LIN {X 0,Y 624.93,Z 1040.405,A -85,B 0,C 180,E1 29774.882,E2 29774.882} C_VEL
LIN {X 0,Y 625.518,Z 1029.116,A -85,B 0,C 180,E1 29772.895,E2 29772.895} C_VEL
LIN {X 0,Y 626.333,Z 1016.12,A -85,B 0,C 180,E1 29770.897,E2 29770.897} C_VEL
LIN {X 0,Y 627.354,Z 1001.616,A -85,B 0,C 180,E1 29768.985,E2 29768.985} C_VEL
LIN {X 0,Y 628.562,Z 986,A -85,B 0,C 180,E1 29767.161,E2 29767.161} C_VEL
LIN {X 0,Y 629.943,Z 968.823,A -85,B 0,C 180,E1 29765.426,E2 29765.426} C_VEL
LIN {X 0,Y 631.502,Z 950.498,A -85,B 0,C 180,E1 29763.784,E2 29763.784} C_VEL
LIN {X 0,Y 633.079,Z 931.694,A -85,B 0,C 180,E1 29762.332,E2 29762.332} C_VEL
LIN {X 0,Y 634.609,Z 913.191,A -85,B 0,C 180,E1 29761.072,E2 29761.072} C_VEL
LIN {X 0,Y 636.354,Z 890.919,A -85,B 0,C 180,E1 29759.762,E2 29759.762} C_VEL
LIN {X 0,Y 637.792,Z 871.802,A -85,B 0,C 180,E1 29758.793,E2 29758.793} C_VEL
LIN {X 0,Y 639.438,Z 848.234,A -85,B 0,C 180,E1 29757.776,E2 29757.776} C_VEL
LIN {X 0,Y 640.692,Z 827.149,A -85,B 0,C 180,E1 29757.025,E2 29757.025} C_VEL
LIN {X 0,Y 641.942,Z 803.825,A -85,B 0,C 180,E1 29756.343,E2 29756.343} C_VEL
LIN {X 0,Y 642.944,Z 779.718,A -85,B 0,C 180,E1 29755.822,E2 29755.822} C_VEL
LIN {X 0,Y 643.646,Z 755.972,A -85,B 0,C 180,E1 29755.448,E2 29755.448} C_VEL
LIN {X 0,Y 647.272,Z 508.069,A -85,B 0,C 180,E1 29752.341,E2 29752.341} C_VEL
LIN {X 0,Y 648.694,Z 406.811,A -85,B 0,C 180,E1 29751.044,E2 29751.044} C_VEL
LIN {X 0,Y 643.579,Z 386.076,A -85,B 0,C 180,E1 29750.391,E2 29750.391} C_VEL
LIN {X 0,Y 636.999,Z 374.634,A -85,B 0,C 180,E1 29749.718,E2 29749.718} C_VEL
LIN {X 0,Y 630.181,Z 356.926,A -85,B 0,C 180,E1 29747.68,E2 29747.68} C_VEL
LIN {X 0,Y 625.657,Z 345.944,A -85,B 0,C 180,E1 29746.338,E2 29746.338} C_VEL
LIN {X 0,Y 624.887,Z 343.395,A -85,B 0,C 180,E1 29746.017,E2 29746.017} C_VEL
LIN {X 0,Y 624.953,Z 343.388,A -85,B 0,C 180,E1 29742.967,E2 29742.967} C_VEL
LIN {X 0,Y 624.886,Z 343.382,A -85,B 0,C 180,E1 29739.963,E2 29739.963} C_VEL
LIN {X 0,Y 624.956,Z 343.376,A -85,B 0,C 180,E1 29736.983,E2 29736.983} C_VEL
LIN {X 0,Y 624.887,Z 343.383,A -85,B 0,C 180,E1 29733.948,E2 29733.948} C_VEL
LIN {X 0,Y 624.955,Z 343.374,A -85,B 0,C 180,E1 29730.903,E2 29730.903} C_VEL
LIN {X 0,Y 624.889,Z 343.378,A -85,B 0,C 180,E1 29727.855,E2 29727.855} C_VEL
LIN {X 0,Y 624.956,Z 343.385,A -85,B 0,C 180,E1 29724.783,E2 29724.783} C_VEL
LIN {X 0,Y 624.887,Z 343.388,A -85,B 0,C 180,E1 29721.791,E2 29721.791} C_VEL
LIN {X 0,Y 624.939,Z 343.372,A -85,B 0,C 180,E1 29718.856,E2 29718.856} C_VEL
LIN {X 0,Y 624.891,Z 343.384,A -85,B 0,C 180,E1 29715.784,E2 29715.784} C_VEL
LIN {X 0,Y 624.92,Z 343.379,A -85,B 0,C 180,E1 29712.944,E2 29712.944} C_VEL
LIN {X 0,Y 624.894,Z 343.373,A -85,B 0,C 180,E1 29709.765,E2 29709.765} C_VEL
LIN {X 0,Y 624.915,Z 343.385,A -85,B 0,C 180,E1 29706.892,E2 29706.892} C_VEL
LIN {X 0,Y 624.896,Z 343.383,A -85,B 0,C 180,E1 29703.67,E2 29703.67} C_VEL
LIN {X 0,Y 624.912,Z 343.384,A -85,B 0,C 180,E1 29700.825,E2 29700.825} C_VEL
LIN {X 0,Y 624.9,Z 343.389,A -85,B 0,C 180,E1 29697.616,E2 29697.616} C_VEL
LIN {X 0,Y 624.907,Z 343.379,A -85,B 0,C 180,E1 29694.767,E2 29694.767} C_VEL
LIN {X 0,Y 624.903,Z 343.389,A -85,B 0,C 180,E1 29691.535,E2 29691.535} C_VEL
LIN {X 0,Y 624.908,Z 343.369,A -85,B 0,C 180,E1 29688.65,E2 29688.65} C_VEL
LIN {X 0,Y 624.904,Z 343.384,A -85,B 0,C 180,E1 29685.451,E2 29685.451} C_VEL
LIN {X 0,Y 624.907,Z 343.38,A -85,B 0,C 180,E1 29682.59,E2 29682.59} C_VEL
LIN {X 0,Y 624.906,Z 343.375,A -85,B 0,C 180,E1 29679.389,E2 29679.389} C_VEL
LIN {X 0,Y 624.899,Z 343.386,A -85,B 0,C 180,E1 29676.62,E2 29676.62} C_VEL
LIN {X 0,Y 624.918,Z 343.387,A -85,B 0,C 180,E1 29673.384,E2 29673.384} C_VEL
LIN {X 0,Y 624.895,Z 343.374,A -85,B 0,C 180,E1 29670.578,E2 29670.578} C_VEL
LIN {X 0,Y 624.941,Z 343.379,A -85,B 0,C 180,E1 29667.478,E2 29667.478} C_VEL
LIN {X 0,Y 624.896,Z 343.387,A -85,B 0,C 180,E1 29664.491,E2 29664.491} C_VEL
LIN {X 0,Y 624.937,Z 343.387,A -85,B 0,C 180,E1 29661.333,E2 29661.333} C_VEL
LIN {X 0,Y 624.896,Z 343.391,A -85,B 0,C 180,E1 29658.391,E2 29658.391} C_VEL
LIN {X 0,Y 624.934,Z 343.351,A -85,B 0,C 180,E1 29655.251,E2 29655.251} C_VEL
LIN {X 0,Y 624.894,Z 343.384,A -85,B 0,C 180,E1 29652.333,E2 29652.333} C_VEL
LIN {X 0,Y 624.953,Z 343.473,A -85,B 0,C 180,E1 29649.73,E2 29649.73} C_VEL
LIN {X 0,Y 626.203,Z 346.794,A -85,B 0,C 180,E1 29649.306,E2 29649.306} C_VEL
LIN {X 0,Y 627.768,Z 350.392,A -85,B 0,C 180,E1 29648.961,E2 29648.961} C_VEL
LIN {X 0,Y 629.852,Z 356.916,A -85,B 0,C 180,E1 29648.631,E2 29648.631} C_VEL
LIN {X 0,Y 633.845,Z 372.513,A -85,B 0,C 180,E1 29648.1,E2 29648.1} C_VEL
LIN {X 0,Y 635.947,Z 377.186,A -85,B 0,C 180,E1 29647.875,E2 29647.875} C_VEL
LIN {X 0,Y 642.615,Z 388.681,A -85,B 0,C 180,E1 29647.223,E2 29647.223} C_VEL
LIN {X 0,Y 638.708,Z 628.744,A -85,B 0,C 180,E1 29644.159,E2 29644.159} C_VEL
LIN {X 0,Y 636.879,Z 738.868,A -85,B 0,C 180,E1 29642.751,E2 29642.751} C_VEL
LIN {X 0,Y 635.934,Z 764.323,A -85,B 0,C 180,E1 29642.266,E2 29642.266} C_VEL
LIN {X 0,Y 634.929,Z 784.357,A -85,B 0,C 180,E1 29641.755,E2 29641.755} C_VEL
LIN {X 0,Y 633.679,Z 806.259,A -85,B 0,C 180,E1 29641.063,E2 29641.063} C_VEL
LIN {X 0,Y 631.998,Z 829.361,A -85,B 0,C 180,E1 29640.154,E2 29640.154} C_VEL
LIN {X 0,Y 630.445,Z 849.976,A -85,B 0,C 180,E1 29639.189,E2 29639.189} C_VEL
LIN {X 0,Y 628.6,Z 871.75,A -85,B 0,C 180,E1 29637.985,E2 29637.985} C_VEL
LIN {X 0,Y 626.972,Z 889.893,A -85,B 0,C 180,E1 29636.829,E2 29636.829} C_VEL
LIN {X 0,Y 625.011,Z 910.955,A -85,B 0,C 180,E1 29635.287,E2 29635.287} C_VEL
LIN {X 0,Y 623.503,Z 927.172,A -85,B 0,C 180,E1 29633.923,E2 29633.923} C_VEL
LIN {X 0,Y 621.814,Z 945.972,A -85,B 0,C 180,E1 29632.146,E2 29632.146} C_VEL
LIN {X 0,Y 620.415,Z 962.253,A -85,B 0,C 180,E1 29630.372,E2 29630.372} C_VEL
LIN {X 0,Y 619.163,Z 977.823,A -85,B 0,C 180,E1 29628.453,E2 29628.453} C_VEL
LIN {X 0,Y 618.189,Z 991.221,A -85,B 0,C 180,E1 29626.539,E2 29626.539} C_VEL
LIN {X 0,Y 617.383,Z 1004.094,A -85,B 0,C 180,E1 29624.443,E2 29624.443} C_VEL
LIN {X 0,Y 616.791,Z 1014.91,A -85,B 0,C 180,E1 29622.356,E2 29622.356} C_VEL
LIN {X 0,Y 616.386,Z 1024.556,A -85,B 0,C 180,E1 29620.184,E2 29620.184} C_VEL
LIN {X 0,Y 616.118,Z 1032.294,A -85,B 0,C 180,E1 29618.023,E2 29618.023} C_VEL
LIN {X 0,Y 616.001,Z 1038.045,A -85,B 0,C 180,E1 29616.056,E2 29616.056} C_VEL
LIN {X 0,Y 615.93,Z 1043.189,A -85,B 0,C 180,E1 29613.723,E2 29613.723} C_VEL
LIN {X 0,Y 615.915,Z 1046.127,A -85,B 0,C 180,E1 29611.768,E2 29611.768} C_VEL
LIN {X 0,Y 615.9,Z 1048.037,A -85,B 0,C 180,E1 29609.628,E2 29609.628} C_VEL
LIN {X 0,Y 615.894,Z 1048.372,A -85,B 0,C 180,E1 29607.395,E2 29607.395} C_VEL
LIN {X 0,Y 615.9,Z 1047.414,A -85,B 0,C 180,E1 29605.423,E2 29605.423} C_VEL
LIN {X 0,Y 615.92,Z 1044.749,A -85,B 0,C 180,E1 29603.1,E2 29603.1} C_VEL
LIN {X 0,Y 615.961,Z 1040.849,A -85,B 0,C 180,E1 29601.035,E2 29601.035} C_VEL
LIN {X 0,Y 616.051,Z 1035.367,A -85,B 0,C 180,E1 29598.864,E2 29598.864} C_VEL
LIN {X 0,Y 616.246,Z 1028.13,A -85,B 0,C 180,E1 29596.679,E2 29596.679} C_VEL
LIN {X 0,Y 616.539,Z 1020.478,A -85,B 0,C 180,E1 29594.768,E2 29594.768} C_VEL
LIN {X 0,Y 617.068,Z 1009.43,A -85,B 0,C 180,E1 29592.459,E2 29592.459} C_VEL
LIN {X 0,Y 617.72,Z 998.488,A -85,B 0,C 180,E1 29590.522,E2 29590.522} C_VEL
LIN {X 0,Y 618.662,Z 984.485,A -85,B 0,C 180,E1 29588.377,E2 29588.377} C_VEL
LIN {X 0,Y 619.676,Z 971.194,A -85,B 0,C 180,E1 29586.613,E2 29586.613} C_VEL
LIN {X 0,Y 621.016,Z 955.276,A -85,B 0,C 180,E1 29584.743,E2 29584.743} C_VEL
LIN {X 0,Y 622.444,Z 938.805,A -85,B 0,C 180,E1 29583.063,E2 29583.063} C_VEL
LIN {X 0,Y 624.226,Z 919.692,A -85,B 0,C 180,E1 29581.332,E2 29581.332} C_VEL
LIN {X 0,Y 625.918,Z 901.36,A -85,B 0,C 180,E1 29579.894,E2 29579.894} C_VEL
LIN {X 0,Y 627.697,Z 882.047,A -85,B 0,C 180,E1 29578.554,E2 29578.554} C_VEL
LIN {X 0,Y 629.506,Z 861.113,A -85,B 0,C 180,E1 29577.313,E2 29577.313} C_VEL
LIN {X 0,Y 631.175,Z 840.831,A -85,B 0,C 180,E1 29576.273,E2 29576.273} C_VEL
LIN {X 0,Y 632.919,Z 817.134,A -85,B 0,C 180,E1 29575.256,E2 29575.256} C_VEL
LIN {X 0,Y 634.242,Z 796.202,A -85,B 0,C 180,E1 29574.511,E2 29574.511} C_VEL
LIN {X 0,Y 635.639,Z 770.4,A -85,B 0,C 180,E1 29573.785,E2 29573.785} C_VEL
LIN {X 0,Y 636.544,Z 749.103,A -85,B 0,C 180,E1 29573.334,E2 29573.334} C_VEL
LIN {X 0,Y 637.275,Z 721.539,A -85,B 0,C 180,E1 29572.919,E2 29572.919} C_VEL
LIN {X 0,Y 641.355,Z 468.268,A -85,B 0,C 180,E1 29569.706,E2 29569.706} C_VEL
LIN {X 0,Y 642.577,Z 388.154,A -85,B 0,C 180,E1 29568.66,E2 29568.66} C_VEL
LIN {X 0,Y 628.337,Z 364.446,A -85,B 0,C 180,E1 29567.206,E2 29567.206} C_VEL
LIN {X 0,Y 619.079,Z 350.106,A -85,B 0,C 180,E1 29566.217,E2 29566.217} C_VEL
LIN {X 0,Y 616.951,Z 344.375,A -85,B 0,C 180,E1 29565.432,E2 29565.432} C_VEL
LIN {X 0,Y 617.017,Z 344.368,A -85,B 0,C 180,E1 29562.357,E2 29562.357} C_VEL
LIN {X 0,Y 616.95,Z 344.369,A -85,B 0,C 180,E1 29559.323,E2 29559.323} C_VEL
LIN {X 0,Y 617.011,Z 344.339,A -85,B 0,C 180,E1 29556.264,E2 29556.264} C_VEL
LIN {X 0,Y 616.951,Z 344.377,A -85,B 0,C 180,E1 29553.216,E2 29553.216} C_VEL
LIN {X 0,Y 617.02,Z 344.373,A -85,B 0,C 180,E1 29550.077,E2 29550.077} C_VEL
LIN {X 0,Y 616.953,Z 344.377,A -85,B 0,C 180,E1 29547.092,E2 29547.092} C_VEL
LIN {X 0,Y 617.012,Z 344.374,A -85,B 0,C 180,E1 29543.938,E2 29543.938} C_VEL
LIN {X 0,Y 616.95,Z 344.37,A -85,B 0,C 180,E1 29540.988,E2 29540.988} C_VEL
LIN {X 0,Y 617.016,Z 344.363,A -85,B 0,C 180,E1 29537.933,E2 29537.933} C_VEL
LIN {X 0,Y 616.95,Z 344.375,A -85,B 0,C 180,E1 29534.933,E2 29534.933} C_VEL
LIN {X 0,Y 617.015,Z 344.374,A -85,B 0,C 180,E1 29531.877,E2 29531.877} C_VEL
LIN {X 0,Y 616.949,Z 344.372,A -85,B 0,C 180,E1 29528.857,E2 29528.857} C_VEL
LIN {X 0,Y 617.016,Z 344.362,A -85,B 0,C 180,E1 29525.86,E2 29525.86} C_VEL
LIN {X 0,Y 616.948,Z 344.376,A -85,B 0,C 180,E1 29522.787,E2 29522.787} C_VEL
LIN {X 0,Y 617.023,Z 344.375,A -85,B 0,C 180,E1 29519.721,E2 29519.721} C_VEL
LIN {X 0,Y 616.947,Z 344.366,A -85,B 0,C 180,E1 29516.655,E2 29516.655} C_VEL
LIN {X 0,Y 617.018,Z 344.361,A -85,B 0,C 180,E1 29513.58,E2 29513.58} C_VEL
LIN {X 0,Y 616.949,Z 344.376,A -85,B 0,C 180,E1 29510.579,E2 29510.579} C_VEL
LIN {X 0,Y 617.014,Z 344.368,A -85,B 0,C 180,E1 29507.553,E2 29507.553} C_VEL
LIN {X 0,Y 616.947,Z 344.364,A -85,B 0,C 180,E1 29504.489,E2 29504.489} C_VEL
LIN {X 0,Y 617.015,Z 344.364,A -85,B 0,C 180,E1 29501.443,E2 29501.443} C_VEL
LIN {X 0,Y 616.948,Z 344.376,A -85,B 0,C 180,E1 29498.414,E2 29498.414} C_VEL
LIN {X 0,Y 617.003,Z 344.37,A -85,B 0,C 180,E1 29495.489,E2 29495.489} C_VEL
LIN {X 0,Y 616.951,Z 344.371,A -85,B 0,C 180,E1 29492.385,E2 29492.385} C_VEL
LIN {X 0,Y 616.989,Z 344.378,A -85,B 0,C 180,E1 29489.519,E2 29489.519} C_VEL
LIN {X 0,Y 616.953,Z 344.378,A -85,B 0,C 180,E1 29486.339,E2 29486.339} C_VEL
LIN {X 0,Y 616.991,Z 344.377,A -85,B 0,C 180,E1 29483.389,E2 29483.389} C_VEL
LIN {X 0,Y 616.956,Z 344.379,A -85,B 0,C 180,E1 29480.316,E2 29480.316} C_VEL
LIN {X 0,Y 616.969,Z 344.367,A -85,B 0,C 180,E1 29477.483,E2 29477.483} C_VEL
LIN {X 0,Y 617.023,Z 344.531,A -85,B 0,C 180,E1 29474.692,E2 29474.692} C_VEL
LIN {X 0,Y 625.556,Z 365.763,A -85,B 0,C 180,E1 29471.99,E2 29471.99} C_VEL
LIN {X 0,Y 629.163,Z 375.222,A -85,B 0,C 180,E1 29470.899,E2 29470.899} C_VEL
LIN {X 0,Y 638.485,Z 391.346,A -85,B 0,C 180,E1 29469.935,E2 29469.935} C_VEL
LIN {X 0,Y 642.629,Z 410.143,A -85,B 0,C 180,E1 29469.355,E2 29469.355} C_VEL
LIN {X 0,Y 638.25,Z 677.094,A -85,B 0,C 180,E1 29465.951,E2 29465.951} C_VEL
LIN {X 0,Y 636.738,Z 767.252,A -85,B 0,C 180,E1 29464.797,E2 29464.797} C_VEL
LIN {X 0,Y 635.766,Z 792.504,A -85,B 0,C 180,E1 29464.317,E2 29464.317} C_VEL
LIN {X 0,Y 634.738,Z 812.614,A -85,B 0,C 180,E1 29463.808,E2 29463.808} C_VEL
LIN {X 0,Y 633.457,Z 835.069,A -85,B 0,C 180,E1 29463.103,E2 29463.103} C_VEL
LIN {X 0,Y 631.844,Z 857.447,A -85,B 0,C 180,E1 29462.229,E2 29462.229} C_VEL
LIN {X 0,Y 630.335,Z 877.622,A -85,B 0,C 180,E1 29461.299,E2 29461.299} C_VEL
LIN {X 0,Y 628.484,Z 900.405,A -85,B 0,C 180,E1 29460.062,E2 29460.062} C_VEL
LIN {X 0,Y 626.885,Z 918.89,A -85,B 0,C 180,E1 29458.9,E2 29458.9} C_VEL
LIN {X 0,Y 625.021,Z 939.869,A -85,B 0,C 180,E1 29457.392,E2 29457.392} C_VEL
LIN {X 0,Y 623.487,Z 957.138,A -85,B 0,C 180,E1 29455.964,E2 29455.964} C_VEL
LIN {X 0,Y 621.967,Z 974.396,A -85,B 0,C 180,E1 29454.353,E2 29454.353} C_VEL
LIN {X 0,Y 620.503,Z 991.086,A -85,B 0,C 180,E1 29452.552,E2 29452.552} C_VEL
LIN {X 0,Y 619.292,Z 1006.237,A -85,B 0,C 180,E1 29450.707,E2 29450.707} C_VEL
LIN {X 0,Y 618.235,Z 1020.607,A -85,B 0,C 180,E1 29448.677,E2 29448.677} C_VEL
LIN {X 0,Y 617.432,Z 1033.123,A -85,B 0,C 180,E1 29446.657,E2 29446.657} C_VEL
LIN {X 0,Y 616.82,Z 1044.181,A -85,B 0,C 180,E1 29444.552,E2 29444.552} C_VEL
LIN {X 0,Y 616.445,Z 1052.774,A -85,B 0,C 180,E1 29442.649,E2 29442.649} C_VEL
LIN {X 0,Y 616.144,Z 1061.604,A -85,B 0,C 180,E1 29440.283,E2 29440.283} C_VEL
LIN {X 0,Y 616.019,Z 1067.49,A -85,B 0,C 180,E1 29438.306,E2 29438.306} C_VEL
LIN {X 0,Y 615.943,Z 1072.696,A -85,B 0,C 180,E1 29436.057,E2 29436.057} C_VEL
LIN {X 0,Y 615.908,Z 1076.01,A -85,B 0,C 180,E1 29433.91,E2 29433.91} C_VEL
LIN {X 0,Y 615.905,Z 1077.836,A -85,B 0,C 180,E1 29431.954,E2 29431.954} C_VEL
LIN {X 0,Y 615.895,Z 1078.417,A -85,B 0,C 180,E1 29429.628,E2 29429.628} C_VEL
LIN {X 0,Y 615.909,Z 1077.495,A -85,B 0,C 180,E1 29427.581,E2 29427.581} C_VEL
LIN {X 0,Y 615.921,Z 1075.085,A -85,B 0,C 180,E1 29425.344,E2 29425.344} C_VEL
LIN {X 0,Y 615.947,Z 1071.102,A -85,B 0,C 180,E1 29423.194,E2 29423.194} C_VEL
LIN {X 0,Y 616.023,Z 1066.219,A -85,B 0,C 180,E1 29421.224,E2 29421.224} C_VEL
LIN {X 0,Y 616.234,Z 1058.661,A -85,B 0,C 180,E1 29418.867,E2 29418.867} C_VEL
LIN {X 0,Y 616.531,Z 1050.749,A -85,B 0,C 180,E1 29416.876,E2 29416.876} C_VEL
LIN {X 0,Y 617.024,Z 1040.404,A -85,B 0,C 180,E1 29414.684,E2 29414.684} C_VEL
LIN {X 0,Y 617.67,Z 1029.115,A -85,B 0,C 180,E1 29412.671,E2 29412.671} C_VEL
LIN {X 0,Y 618.548,Z 1016.119,A -85,B 0,C 180,E1 29410.647,E2 29410.647} C_VEL
LIN {X 0,Y 619.65,Z 1001.614,A -85,B 0,C 180,E1 29408.711,E2 29408.711} C_VEL
LIN {X 0,Y 620.977,Z 985.782,A -85,B 0,C 180,E1 29406.842,E2 29406.842} C_VEL
LIN {X 0,Y 622.442,Z 968.822,A -85,B 0,C 180,E1 29405.11,E2 29405.11} C_VEL
LIN {X 0,Y 623.88,Z 952.658,A -85,B 0,C 180,E1 29403.644,E2 29403.644} C_VEL
LIN {X 0,Y 625.655,Z 932.82,A -85,B 0,C 180,E1 29402.079,E2 29402.079} C_VEL
LIN {X 0,Y 627.208,Z 915.193,A -85,B 0,C 180,E1 29400.855,E2 29400.855} C_VEL
LIN {X 0,Y 629.064,Z 893.416,A -85,B 0,C 180,E1 29399.533,E2 29399.533} C_VEL
LIN {X 0,Y 630.661,Z 873.465,A -85,B 0,C 180,E1 29398.499,E2 29398.499} C_VEL
LIN {X 0,Y 632.318,Z 851.795,A -85,B 0,C 180,E1 29397.53,E2 29397.53} C_VEL
LIN {X 0,Y 633.817,Z 828.417,A -85,B 0,C 180,E1 29396.675,E2 29396.675} C_VEL
LIN {X 0,Y 635.037,Z 807.046,A -85,B 0,C 180,E1 29396.035,E2 29396.035} C_VEL
LIN {X 0,Y 636.223,Z 781.484,A -85,B 0,C 180,E1 29395.452,E2 29395.452} C_VEL
LIN {X 0,Y 636.947,Z 759.346,A -85,B 0,C 180,E1 29395.09,E2 29395.09} C_VEL
LIN {X 0,Y 640.743,Z 518.127,A -85,B 0,C 180,E1 29392.034,E2 29392.034} C_VEL
LIN {X 0,Y 642.4,Z 408.639,A -85,B 0,C 180,E1 29390.624,E2 29390.624} C_VEL
LIN {X 0,Y 637.907,Z 390.365,A -85,B 0,C 180,E1 29390.04,E2 29390.04} C_VEL
LIN {X 0,Y 628.778,Z 374.728,A -85,B 0,C 180,E1 29389.126,E2 29389.126} C_VEL
LIN {X 0,Y 620.891,Z 354.378,A -85,B 0,C 180,E1 29386.711,E2 29386.711} C_VEL
LIN {X 0,Y 616.988,Z 344.415,A -85,B 0,C 180,E1 29385.47,E2 29385.47} C_VEL
LIN {X 0,Y 616.953,Z 344.382,A -85,B 0,C 180,E1 29382.267,E2 29382.267} C_VEL
LIN {X 0,Y 616.974,Z 344.369,A -85,B 0,C 180,E1 29379.442,E2 29379.442} C_VEL
LIN {X 0,Y 616.959,Z 344.381,A -85,B 0,C 180,E1 29376.267,E2 29376.267} C_VEL
LIN {X 0,Y 616.967,Z 344.37,A -85,B 0,C 180,E1 29373.422,E2 29373.422} C_VEL
LIN {X 0,Y 616.959,Z 344.375,A -85,B 0,C 180,E1 29370.16,E2 29370.16} C_VEL
LIN {X 0,Y 616.964,Z 344.364,A -85,B 0,C 180,E1 29367.362,E2 29367.362} C_VEL
LIN {X 0,Y 616.962,Z 344.366,A -85,B 0,C 180,E1 29364.105,E2 29364.105} C_VEL
LIN {X 0,Y 616.964,Z 344.374,A -85,B 0,C 180,E1 29361.27,E2 29361.27} C_VEL
LIN {X 0,Y 616.961,Z 344.376,A -85,B 0,C 180,E1 29357.949,E2 29357.949} C_VEL
LIN {X 0,Y 616.976,Z 344.369,A -85,B 0,C 180,E1 29355.029,E2 29355.029} C_VEL
LIN {X 0,Y 616.957,Z 344.377,A -85,B 0,C 180,E1 29351.783,E2 29351.783} C_VEL
LIN {X 0,Y 616.981,Z 344.358,A -85,B 0,C 180,E1 29348.856,E2 29348.856} C_VEL
LIN {X 0,Y 616.956,Z 344.369,A -85,B 0,C 180,E1 29345.674,E2 29345.674} C_VEL
LIN {X 0,Y 616.99,Z 344.368,A -85,B 0,C 180,E1 29342.694,E2 29342.694} C_VEL
LIN {X 0,Y 616.953,Z 344.359,A -85,B 0,C 180,E1 29339.525,E2 29339.525} C_VEL
LIN {X 0,Y 616.993,Z 344.373,A -85,B 0,C 180,E1 29336.562,E2 29336.562} C_VEL
LIN {X 0,Y 616.952,Z 344.369,A -85,B 0,C 180,E1 29333.392,E2 29333.392} C_VEL
LIN {X 0,Y 616.992,Z 344.373,A -85,B 0,C 180,E1 29330.485,E2 29330.485} C_VEL
LIN {X 0,Y 616.956,Z 344.377,A -85,B 0,C 180,E1 29327.33,E2 29327.33} C_VEL
LIN {X 0,Y 616.979,Z 344.368,A -85,B 0,C 180,E1 29324.49,E2 29324.49} C_VEL
LIN {X 0,Y 616.961,Z 344.377,A -85,B 0,C 180,E1 29321.283,E2 29321.283} C_VEL
LIN {X 0,Y 616.977,Z 344.362,A -85,B 0,C 180,E1 29318.415,E2 29318.415} C_VEL
LIN {X 0,Y 616.959,Z 344.363,A -85,B 0,C 180,E1 29315.173,E2 29315.173} C_VEL
LIN {X 0,Y 616.987,Z 344.374,A -85,B 0,C 180,E1 29312.233,E2 29312.233} C_VEL
LIN {X 0,Y 616.961,Z 344.379,A -85,B 0,C 180,E1 29309.086,E2 29309.086} C_VEL
LIN {X 0,Y 616.988,Z 344.363,A -85,B 0,C 180,E1 29306.118,E2 29306.118} C_VEL
LIN {X 0,Y 616.958,Z 344.372,A -85,B 0,C 180,E1 29302.922,E2 29302.922} C_VEL
LIN {X 0,Y 616.984,Z 344.368,A -85,B 0,C 180,E1 29300.045,E2 29300.045} C_VEL
LIN {X 0,Y 616.958,Z 344.354,A -85,B 0,C 180,E1 29296.828,E2 29296.828} C_VEL
LIN {X 0,Y 617.003,Z 344.371,A -85,B 0,C 180,E1 29293.787,E2 29293.787} C_VEL
LIN {X 0,Y 616.958,Z 344.381,A -85,B 0,C 180,E1 29290.656,E2 29290.656} C_VEL
LIN {X 0,Y 616.962,Z 344.424,A -85,B 0,C 180,E1 29290.312,E2 29290.312} C_VEL
LIN {X 0,Y 619.286,Z 350.473,A -85,B 0,C 180,E1 29289.559,E2 29289.559} C_VEL
LIN {X 0,Y 635.41,Z 376.25,A -85,B 0,C 180,E1 29287.929,E2 29287.929} C_VEL
LIN {X 0,Y 635.947,Z 377.186,A -85,B 0,C 180,E1 29287.875,E2 29287.875} C_VEL
LIN {X 0,Y 637.696,Z 381.876,A -85,B 0,C 180,E1 29287.678,E2 29287.678} C_VEL
LIN {X 0,Y 638.342,Z 388.319,A -85,B 0,C 180,E1 29287.539,E2 29287.539} C_VEL
LIN {X 0,Y 637.479,Z 398.608,A -85,B 0,C 180,E1 29287.456,E2 29287.456} C_VEL
LIN {X 0,Y 636.01,Z 411.557,A -85,B 0,C 180,E1 29287.379,E2 29287.379} C_VEL
LIN {X 0,Y 635.973,Z 412.733,A -85,B 0,C 180,E1 29287.365,E2 29287.365} C_VEL
LIN {X 0,Y 631.746,Z 660.219,A -85,B 0,C 180,E1 29284.189,E2 29284.189} C_VEL
LIN {X 0,Y 630.304,Z 739.834,A -85,B 0,C 180,E1 29283.154,E2 29283.154} C_VEL
LIN {X 0,Y 629.304,Z 764.933,A -85,B 0,C 180,E1 29282.668,E2 29282.668} C_VEL
LIN {X 0,Y 628.251,Z 784.817,A -85,B 0,C 180,E1 29282.156,E2 29282.156} C_VEL
LIN {X 0,Y 626.858,Z 807.75,A -85,B 0,C 180,E1 29281.419,E2 29281.419} C_VEL
LIN {X 0,Y 625.122,Z 830.21,A -85,B 0,C 180,E1 29280.52,E2 29280.52} C_VEL
LIN {X 0,Y 623.405,Z 851.74,A -85,B 0,C 180,E1 29279.499,E2 29279.499} C_VEL
LIN {X 0,Y 621.518,Z 872.423,A -85,B 0,C 180,E1 29278.333,E2 29278.333} C_VEL
LIN {X 0,Y 619.797,Z 890.524,A -85,B 0,C 180,E1 29277.165,E2 29277.165} C_VEL
LIN {X 0,Y 617.646,Z 912.113,A -85,B 0,C 180,E1 29275.558,E2 29275.558} C_VEL
LIN {X 0,Y 616.012,Z 928.638,A -85,B 0,C 180,E1 29274.144,E2 29274.144} C_VEL
LIN {X 0,Y 614.23,Z 946.758,A -85,B 0,C 180,E1 29272.386,E2 29272.386} C_VEL
LIN {X 0,Y 612.691,Z 963.333,A -85,B 0,C 180,E1 29270.541,E2 29270.541} C_VEL
LIN {X 0,Y 611.24,Z 980.108,A -85,B 0,C 180,E1 29268.404,E2 29268.404} C_VEL
LIN {X 0,Y 610.279,Z 992.662,A -85,B 0,C 180,E1 29266.564,E2 29266.564} C_VEL
LIN {X 0,Y 609.399,Z 1005.783,A -85,B 0,C 180,E1 29264.345,E2 29264.345} C_VEL
LIN {X 0,Y 608.841,Z 1015.497,A -85,B 0,C 180,E1 29262.424,E2 29262.424} C_VEL
LIN {X 0,Y 608.41,Z 1025.019,A -85,B 0,C 180,E1 29260.224,E2 29260.224} C_VEL
LIN {X 0,Y 608.139,Z 1032.381,A -85,B 0,C 180,E1 29258.129,E2 29258.129} C_VEL
LIN {X 0,Y 608.012,Z 1038.118,A -85,B 0,C 180,E1 29256.136,E2 29256.136} C_VEL
LIN {X 0,Y 607.934,Z 1043.234,A -85,B 0,C 180,E1 29253.772,E2 29253.772} C_VEL
LIN {X 0,Y 607.916,Z 1046.159,A -85,B 0,C 180,E1 29251.791,E2 29251.791} C_VEL
LIN {X 0,Y 607.901,Z 1048.057,A -85,B 0,C 180,E1 29249.623,E2 29249.623} C_VEL
LIN {X 0,Y 607.894,Z 1048.365,A -85,B 0,C 180,E1 29247.36,E2 29247.36} C_VEL
LIN {X 0,Y 607.899,Z 1047.404,A -85,B 0,C 180,E1 29245.377,E2 29245.377} C_VEL
LIN {X 0,Y 607.921,Z 1044.704,A -85,B 0,C 180,E1 29243.009,E2 29243.009} C_VEL
LIN {X 0,Y 607.97,Z 1040.79,A -85,B 0,C 180,E1 29240.916,E2 29240.916} C_VEL
LIN {X 0,Y 608.075,Z 1035.293,A -85,B 0,C 180,E1 29238.716,E2 29238.716} C_VEL
LIN {X 0,Y 608.286,Z 1028.026,A -85,B 0,C 180,E1 29236.502,E2 29236.502} C_VEL
LIN {X 0,Y 608.599,Z 1020.359,A -85,B 0,C 180,E1 29234.564,E2 29234.564} C_VEL
LIN {X 0,Y 609.176,Z 1009.276,A -85,B 0,C 180,E1 29232.224,E2 29232.224} C_VEL
LIN {X 0,Y 609.848,Z 998.896,A -85,B 0,C 180,E1 29230.36,E2 29230.36} C_VEL
LIN {X 0,Y 610.811,Z 985.692,A -85,B 0,C 180,E1 29228.287,E2 29228.287} C_VEL
LIN {X 0,Y 611.938,Z 971.742,A -85,B 0,C 180,E1 29226.402,E2 29226.402} C_VEL
LIN {X 0,Y 613.377,Z 955.934,A -85,B 0,C 180,E1 29224.51,E2 29224.51} C_VEL
LIN {X 0,Y 615.013,Z 938.663,A -85,B 0,C 180,E1 29222.711,E2 29222.711} C_VEL
LIN {X 0,Y 616.794,Z 921.137,A -85,B 0,C 180,E1 29221.093,E2 29221.093} C_VEL
LIN {X 0,Y 618.683,Z 901.859,A -85,B 0,C 180,E1 29219.558,E2 29219.558} C_VEL
LIN {X 0,Y 620.572,Z 882.575,A -85,B 0,C 180,E1 29218.205,E2 29218.205} C_VEL
LIN {X 0,Y 622.515,Z 861.552,A -85,B 0,C 180,E1 29216.945,E2 29216.945} C_VEL
LIN {X 0,Y 624.171,Z 842.465,A -85,B 0,C 180,E1 29215.952,E2 29215.952} C_VEL
LIN {X 0,Y 626.019,Z 819.2,A -85,B 0,C 180,E1 29214.928,E2 29214.928} C_VEL
LIN {X 0,Y 627.409,Z 798.552,A -85,B 0,C 180,E1 29214.177,E2 29214.177} C_VEL
LIN {X 0,Y 628.81,Z 774.942,A -85,B 0,C 180,E1 29213.476,E2 29213.476} C_VEL
LIN {X 0,Y 629.874,Z 751.394,A -85,B 0,C 180,E1 29212.958,E2 29212.958} C_VEL
LIN {X 0,Y 630.648,Z 727.106,A -85,B 0,C 180,E1 29212.57,E2 29212.57} C_VEL
LIN {X 0,Y 635.022,Z 474.062,A -85,B 0,C 180,E1 29209.328,E2 29209.328} C_VEL
LIN {X 0,Y 636.398,Z 391.316,A -85,B 0,C 180,E1 29208.238,E2 29208.238} C_VEL
LIN {X 0,Y 623.168,Z 369.368,A -85,B 0,C 180,E1 29206.858,E2 29206.858} C_VEL
LIN {X 0,Y 612.17,Z 352.556,A -85,B 0,C 180,E1 29205.66,E2 29205.66} C_VEL
LIN {X 0,Y 610.765,Z 350.187,A -85,B 0,C 180,E1 29205.477,E2 29205.477} C_VEL
LIN {X 0,Y 609.052,Z 345.365,A -85,B 0,C 180,E1 29204.803,E2 29204.803} C_VEL
LIN {X 0,Y 609.018,Z 345.347,A -85,B 0,C 180,E1 29201.667,E2 29201.667} C_VEL
LIN {X 0,Y 609.049,Z 345.361,A -85,B 0,C 180,E1 29198.719,E2 29198.719} C_VEL
LIN {X 0,Y 609.014,Z 345.33,A -85,B 0,C 180,E1 29195.535,E2 29195.535} C_VEL
LIN {X 0,Y 609.056,Z 345.365,A -85,B 0,C 180,E1 29192.58,E2 29192.58} C_VEL
LIN {X 0,Y 609.018,Z 345.364,A -85,B 0,C 180,E1 29189.4,E2 29189.4} C_VEL
LIN {X 0,Y 609.062,Z 345.365,A -85,B 0,C 180,E1 29186.417,E2 29186.417} C_VEL
LIN {X 0,Y 609.017,Z 345.365,A -85,B 0,C 180,E1 29183.308,E2 29183.308} C_VEL
LIN {X 0,Y 609.054,Z 345.361,A -85,B 0,C 180,E1 29180.368,E2 29180.368} C_VEL
LIN {X 0,Y 609.013,Z 345.36,A -85,B 0,C 180,E1 29177.149,E2 29177.149} C_VEL
LIN {X 0,Y 609.066,Z 345.353,A -85,B 0,C 180,E1 29174.159,E2 29174.159} C_VEL
LIN {X 0,Y 609.015,Z 345.363,A -85,B 0,C 180,E1 29171.075,E2 29171.075} C_VEL
LIN {X 0,Y 609.069,Z 345.365,A -85,B 0,C 180,E1 29168.021,E2 29168.021} C_VEL
LIN {X 0,Y 609.01,Z 345.359,A -85,B 0,C 180,E1 29164.898,E2 29164.898} C_VEL
LIN {X 0,Y 609.068,Z 345.352,A -85,B 0,C 180,E1 29161.882,E2 29161.882} C_VEL
LIN {X 0,Y 609.012,Z 345.365,A -85,B 0,C 180,E1 29158.777,E2 29158.777} C_VEL
LIN {X 0,Y 609.075,Z 345.361,A -85,B 0,C 180,E1 29155.669,E2 29155.669} C_VEL
LIN {X 0,Y 609.008,Z 345.352,A -85,B 0,C 180,E1 29152.598,E2 29152.598} C_VEL
LIN {X 0,Y 609.075,Z 345.351,A -85,B 0,C 180,E1 29149.53,E2 29149.53} C_VEL
LIN {X 0,Y 609.01,Z 345.366,A -85,B 0,C 180,E1 29146.421,E2 29146.421} C_VEL
LIN {X 0,Y 609.077,Z 345.357,A -85,B 0,C 180,E1 29143.402,E2 29143.402} C_VEL
LIN {X 0,Y 609.007,Z 345.352,A -85,B 0,C 180,E1 29140.331,E2 29140.331} C_VEL
LIN {X 0,Y 609.082,Z 345.35,A -85,B 0,C 180,E1 29137.307,E2 29137.307} C_VEL
LIN {X 0,Y 609.01,Z 345.366,A -85,B 0,C 180,E1 29134.209,E2 29134.209} C_VEL
LIN {X 0,Y 609.077,Z 345.361,A -85,B 0,C 180,E1 29131.045,E2 29131.045} C_VEL
LIN {X 0,Y 609.009,Z 345.367,A -85,B 0,C 180,E1 29128.084,E2 29128.084} C_VEL
LIN {X 0,Y 609.076,Z 345.363,A -85,B 0,C 180,E1 29125.003,E2 29125.003} C_VEL
LIN {X 0,Y 609.008,Z 345.366,A -85,B 0,C 180,E1 29121.998,E2 29121.998} C_VEL
LIN {X 0,Y 609.08,Z 345.362,A -85,B 0,C 180,E1 29118.896,E2 29118.896} C_VEL
LIN {X 0,Y 609.011,Z 345.369,A -85,B 0,C 180,E1 29115.847,E2 29115.847} C_VEL
LIN {X 0,Y 609.071,Z 345.565,A -85,B 0,C 180,E1 29115.328,E2 29115.328} C_VEL
LIN {X 0,Y 617.648,Z 366.692,A -85,B 0,C 180,E1 29112.558,E2 29112.558} C_VEL
LIN {X 0,Y 620.898,Z 374.872,A -85,B 0,C 180,E1 29111.58,E2 29111.58} C_VEL
LIN {X 0,Y 632.845,Z 395.363,A -85,B 0,C 180,E1 29110.311,E2 29110.311} C_VEL
LIN {X 0,Y 636.439,Z 411.894,A -85,B 0,C 180,E1 29109.793,E2 29109.793} C_VEL
LIN {X 0,Y 631.746,Z 678.208,A -85,B 0,C 180,E1 29106.362,E2 29106.362} C_VEL
LIN {X 0,Y 630.151,Z 767.053,A -85,B 0,C 180,E1 29105.214,E2 29105.214} C_VEL
LIN {X 0,Y 629.116,Z 792.394,A -85,B 0,C 180,E1 29104.729,E2 29104.729} C_VEL
LIN {X 0,Y 628.015,Z 812.716,A -85,B 0,C 180,E1 29104.21,E2 29104.21} C_VEL
LIN {X 0,Y 626.572,Z 836.174,A -85,B 0,C 180,E1 29103.46,E2 29103.46} C_VEL
LIN {X 0,Y 624.875,Z 858.359,A -85,B 0,C 180,E1 29102.578,E2 29102.578} C_VEL
LIN {X 0,Y 623.131,Z 880.429,A -85,B 0,C 180,E1 29101.541,E2 29101.541} C_VEL
LIN {X 0,Y 621.251,Z 901.593,A -85,B 0,C 180,E1 29100.356,E2 29100.356} C_VEL
LIN {X 0,Y 619.546,Z 920.145,A -85,B 0,C 180,E1 29099.17,E2 29099.17} C_VEL
LIN {X 0,Y 617.49,Z 941.596,A -85,B 0,C 180,E1 29097.588,E2 29097.588} C_VEL
LIN {X 0,Y 615.939,Z 958.032,A -85,B 0,C 180,E1 29096.203,E2 29096.203} C_VEL
LIN {X 0,Y 614.202,Z 976.677,A -85,B 0,C 180,E1 29094.425,E2 29094.425} C_VEL
LIN {X 0,Y 612.845,Z 991.46,A -85,B 0,C 180,E1 29092.804,E2 29092.804} C_VEL
LIN {X 0,Y 611.522,Z 1006.997,A -85,B 0,C 180,E1 29090.882,E2 29090.882} C_VEL
LIN {X 0,Y 610.387,Z 1021.24,A -85,B 0,C 180,E1 29088.827,E2 29088.827} C_VEL
LIN {X 0,Y 609.532,Z 1033.689,A -85,B 0,C 180,E1 29086.781,E2 29086.781} C_VEL
LIN {X 0,Y 608.878,Z 1044.639,A -85,B 0,C 180,E1 29084.649,E2 29084.649} C_VEL
LIN {X 0,Y 608.463,Z 1053.583,A -85,B 0,C 180,E1 29082.624,E2 29082.624} C_VEL
LIN {X 0,Y 608.158,Z 1061.907,A -85,B 0,C 180,E1 29080.324,E2 29080.324} C_VEL
LIN {X 0,Y 608.023,Z 1067.491,A -85,B 0,C 180,E1 29078.416,E2 29078.416} C_VEL
LIN {X 0,Y 607.945,Z 1072.696,A -85,B 0,C 180,E1 29076.137,E2 29076.137} C_VEL
LIN {X 0,Y 607.909,Z 1076.009,A -85,B 0,C 180,E1 29073.961,E2 29073.961} C_VEL
LIN {X 0,Y 607.906,Z 1077.836,A -85,B 0,C 180,E1 29071.979,E2 29071.979} C_VEL
LIN {X 0,Y 607.895,Z 1078.417,A -85,B 0,C 180,E1 29069.623,E2 29069.623} C_VEL
LIN {X 0,Y 607.908,Z 1077.495,A -85,B 0,C 180,E1 29067.549,E2 29067.549} C_VEL
LIN {X 0,Y 607.923,Z 1075.085,A -85,B 0,C 180,E1 29065.283,E2 29065.283} C_VEL
LIN {X 0,Y 607.957,Z 1071.102,A -85,B 0,C 180,E1 29063.104,E2 29063.104} C_VEL
LIN {X 0,Y 608.035,Z 1066.219,A -85,B 0,C 180,E1 29061.108,E2 29061.108} C_VEL
LIN {X 0,Y 608.266,Z 1058.66,A -85,B 0,C 180,E1 29058.719,E2 29058.719} C_VEL
LIN {X 0,Y 608.588,Z 1050.748,A -85,B 0,C 180,E1 29056.702,E2 29056.702} C_VEL
LIN {X 0,Y 609.123,Z 1040.402,A -85,B 0,C 180,E1 29054.48,E2 29054.48} C_VEL
LIN {X 0,Y 609.827,Z 1029.113,A -85,B 0,C 180,E1 29052.441,E2 29052.441} C_VEL
LIN {X 0,Y 610.779,Z 1016.117,A -85,B 0,C 180,E1 29050.391,E2 29050.391} C_VEL
LIN {X 0,Y 611.957,Z 1001.612,A -85,B 0,C 180,E1 29048.43,E2 29048.43} C_VEL
LIN {X 0,Y 613.372,Z 985.999,A -85,B 0,C 180,E1 29046.562,E2 29046.562} C_VEL
LIN {X 0,Y 614.907,Z 968.972,A -85,B 0,C 180,E1 29044.813,E2 29044.813} C_VEL
LIN {X 0,Y 616.661,Z 950.759,A -85,B 0,C 180,E1 29043.155,E2 29043.155} C_VEL
LIN {X 0,Y 618.487,Z 931.255,A -85,B 0,C 180,E1 29041.621,E2 29041.621} C_VEL
LIN {X 0,Y 620.297,Z 912.013,A -85,B 0,C 180,E1 29040.286,E2 29040.286} C_VEL
LIN {X 0,Y 622.247,Z 890.482,A -85,B 0,C 180,E1 29039.002,E2 29039.002} C_VEL
LIN {X 0,Y 623.869,Z 871.366,A -85,B 0,C 180,E1 29038.015,E2 29038.015} C_VEL
LIN {X 0,Y 625.724,Z 847.82,A -85,B 0,C 180,E1 29036.982,E2 29036.982} C_VEL
LIN {X 0,Y 627.182,Z 825.971,A -85,B 0,C 180,E1 29036.193,E2 29036.193} C_VEL
LIN {X 0,Y 628.648,Z 801.827,A -85,B 0,C 180,E1 29035.49,E2 29035.49} C_VEL
LIN {X 0,Y 629.71,Z 779.15,A -85,B 0,C 180,E1 29034.997,E2 29034.997} C_VEL
LIN {X 0,Y 630.482,Z 755.478,A -85,B 0,C 180,E1 29034.619,E2 29034.619} C_VEL
LIN {X 0,Y 634.576,Z 507.829,A -85,B 0,C 180,E1 29031.462,E2 29031.462} C_VEL
LIN {X 0,Y 636.13,Z 410.472,A -85,B 0,C 180,E1 29030.196,E2 29030.196} C_VEL
LIN {X 0,Y 632.258,Z 394.616,A -85,B 0,C 180,E1 29029.682,E2 29029.682} C_VEL
LIN {X 0,Y 620.448,Z 374.384,A -85,B 0,C 180,E1 29028.467,E2 29028.467} C_VEL
LIN {X 0,Y 612.728,Z 354.981,A -85,B 0,C 180,E1 29026.089,E2 29026.089} C_VEL
LIN {X 0,Y 609.065,Z 345.367,A -85,B 0,C 180,E1 29024.867,E2 29024.867} C_VEL
LIN {X 0,Y 609.009,Z 345.37,A -85,B 0,C 180,E1 29021.93,E2 29021.93} C_VEL
LIN {X 0,Y 609.077,Z 345.362,A -85,B 0,C 180,E1 29018.837,E2 29018.837} C_VEL
LIN {X 0,Y 609.012,Z 345.368,A -85,B 0,C 180,E1 29015.767,E2 29015.767} C_VEL
LIN {X 0,Y 609.057,Z 345.366,A -85,B 0,C 180,E1 29012.58,E2 29012.58} C_VEL
LIN {X 0,Y 609.014,Z 345.363,A -85,B 0,C 180,E1 29009.616,E2 29009.616} C_VEL
LIN {X 0,Y 609.062,Z 345.353,A -85,B 0,C 180,E1 29006.522,E2 29006.522} C_VEL
LIN {X 0,Y 609.009,Z 345.353,A -85,B 0,C 180,E1 29003.616,E2 29003.616} C_VEL
LIN {X 0,Y 609.076,Z 345.362,A -85,B 0,C 180,E1 29000.568,E2 29000.568} C_VEL
LIN {X 0,Y 609.011,Z 345.364,A -85,B 0,C 180,E1 28997.485,E2 28997.485} C_VEL
LIN {X 0,Y 609.07,Z 345.348,A -85,B 0,C 180,E1 28994.353,E2 28994.353} C_VEL
LIN {X 0,Y 609.012,Z 345.364,A -85,B 0,C 180,E1 28991.363,E2 28991.363} C_VEL
LIN {X 0,Y 609.064,Z 345.355,A -85,B 0,C 180,E1 28988.211,E2 28988.211} C_VEL
LIN {X 0,Y 609.012,Z 345.356,A -85,B 0,C 180,E1 28985.275,E2 28985.275} C_VEL
LIN {X 0,Y 609.069,Z 345.364,A -85,B 0,C 180,E1 28982.164,E2 28982.164} C_VEL
LIN {X 0,Y 609.011,Z 345.346,A -85,B 0,C 180,E1 28979.153,E2 28979.153} C_VEL
LIN {X 0,Y 609.068,Z 345.363,A -85,B 0,C 180,E1 28976.046,E2 28976.046} C_VEL
LIN {X 0,Y 609.014,Z 345.357,A -85,B 0,C 180,E1 28973.022,E2 28973.022} C_VEL
LIN {X 0,Y 609.06,Z 345.352,A -85,B 0,C 180,E1 28969.883,E2 28969.883} C_VEL
LIN {X 0,Y 609.016,Z 345.364,A -85,B 0,C 180,E1 28966.905,E2 28966.905} C_VEL
LIN {X 0,Y 609.062,Z 345.349,A -85,B 0,C 180,E1 28963.794,E2 28963.794} C_VEL
LIN {X 0,Y 609.017,Z 345.363,A -85,B 0,C 180,E1 28960.83,E2 28960.83} C_VEL
LIN {X 0,Y 609.072,Z 345.357,A -85,B 0,C 180,E1 28957.714,E2 28957.714} C_VEL
LIN {X 0,Y 609.013,Z 345.35,A -85,B 0,C 180,E1 28954.731,E2 28954.731} C_VEL
LIN {X 0,Y 609.064,Z 345.357,A -85,B 0,C 180,E1 28951.57,E2 28951.57} C_VEL
LIN {X 0,Y 609.017,Z 345.366,A -85,B 0,C 180,E1 28948.621,E2 28948.621} C_VEL
LIN {X 0,Y 609.065,Z 345.36,A -85,B 0,C 180,E1 28945.5,E2 28945.5} C_VEL
LIN {X 0,Y 609.018,Z 345.364,A -85,B 0,C 180,E1 28942.466,E2 28942.466} C_VEL
LIN {X 0,Y 609.061,Z 345.36,A -85,B 0,C 180,E1 28939.326,E2 28939.326} C_VEL
LIN {X 0,Y 609.015,Z 345.332,A -85,B 0,C 180,E1 28936.389,E2 28936.389} C_VEL
LIN {X 0,Y 609.059,Z 345.368,A -85,B 0,C 180,E1 28933.203,E2 28933.203} C_VEL
LIN {X 0,Y 609.062,Z 345.576,A -85,B 0,C 180,E1 28930.887,E2 28930.887} C_VEL
LIN {X 0,Y 611.013,Z 350.763,A -85,B 0,C 180,E1 28930.235,E2 28930.235} C_VEL
LIN {X 0,Y 626.828,Z 375.591,A -85,B 0,C 180,E1 28928.59,E2 28928.59} C_VEL
LIN {X 0,Y 636.341,Z 391.797,A -85,B 0,C 180,E1 28927.637,E2 28927.637} C_VEL
LIN {X 0,Y 635.973,Z 412.733,A -85,B 0,C 180,E1 28927.365,E2 28927.365} C_VEL
LIN {X 0,Y 635.047,Z 420.433,A -85,B 0,C 180,E1 28927.323,E2 28927.323} C_VEL
LIN {X 0,Y 629.815,Z 441.007,A -85,B 0,C 180,E1 28927.413,E2 28927.413} C_VEL
LIN {X 0,Y 629.133,Z 447.61,A -85,B 0,C 180,E1 28927.368,E2 28927.368} C_VEL
LIN {X 0,Y 624.619,Z 699.187,A -85,B 0,C 180,E1 28924.124,E2 28924.124} C_VEL
LIN {X 0,Y 623.697,Z 743.497,A -85,B 0,C 180,E1 28923.524,E2 28923.524} C_VEL
LIN {X 0,Y 622.627,Z 767.01,A -85,B 0,C 180,E1 28923.044,E2 28923.044} C_VEL
LIN {X 0,Y 621.497,Z 787.189,A -85,B 0,C 180,E1 28922.51,E2 28922.51} C_VEL
LIN {X 0,Y 619.803,Z 812.008,A -85,B 0,C 180,E1 28921.676,E2 28921.676} C_VEL
LIN {X 0,Y 618.178,Z 832.167,A -85,B 0,C 180,E1 28920.847,E2 28920.847} C_VEL
LIN {X 0,Y 616.198,Z 855.203,A -85,B 0,C 180,E1 28919.718,E2 28919.718} C_VEL
LIN {X 0,Y 614.304,Z 874.686,A -85,B 0,C 180,E1 28918.59,E2 28918.59} C_VEL
LIN {X 0,Y 612.292,Z 894.753,A -85,B 0,C 180,E1 28917.262,E2 28917.262} C_VEL
LIN {X 0,Y 610.169,Z 914.461,A -85,B 0,C 180,E1 28915.738,E2 28915.738} C_VEL
LIN {X 0,Y 608.261,Z 932.973,A -85,B 0,C 180,E1 28914.11,E2 28914.11} C_VEL
LIN {X 0,Y 606.372,Z 950.537,A -85,B 0,C 180,E1 28912.32,E2 28912.32} C_VEL
LIN {X 0,Y 604.843,Z 966.182,A -85,B 0,C 180,E1 28910.516,E2 28910.516} C_VEL
LIN {X 0,Y 603.374,Z 981.698,A -85,B 0,C 180,E1 28908.452,E2 28908.452} C_VEL
LIN {X 0,Y 602.275,Z 995.359,A -85,B 0,C 180,E1 28906.393,E2 28906.393} C_VEL
LIN {X 0,Y 601.407,Z 1007.51,A -85,B 0,C 180,E1 28904.236,E2 28904.236} C_VEL
LIN {X 0,Y 600.8,Z 1017.904,A -85,B 0,C 180,E1 28902.105,E2 28902.105} C_VEL
LIN {X 0,Y 600.376,Z 1026.879,A -85,B 0,C 180,E1 28899.877,E2 28899.877} C_VEL
LIN {X 0,Y 600.123,Z 1033.674,A -85,B 0,C 180,E1 28897.852,E2 28897.852} C_VEL
LIN {X 0,Y 599.975,Z 1040.012,A -85,B 0,C 180,E1 28895.451,E2 28895.451} C_VEL
LIN {X 0,Y 599.921,Z 1043.917,A -85,B 0,C 180,E1 28893.44,E2 28893.44} C_VEL
LIN {X 0,Y 599.913,Z 1046.869,A -85,B 0,C 180,E1 28891.242,E2 28891.242} C_VEL
LIN {X 0,Y 599.909,Z 1048.271,A -85,B 0,C 180,E1 28888.949,E2 28888.949} C_VEL
LIN {X 0,Y 599.907,Z 1048.267,A -85,B 0,C 180,E1 28886.943,E2 28886.943} C_VEL
LIN {X 0,Y 599.914,Z 1046.729,A -85,B 0,C 180,E1 28884.548,E2 28884.548} C_VEL
LIN {X 0,Y 599.92,Z 1043.857,A -85,B 0,C 180,E1 28882.434,E2 28882.434} C_VEL
LIN {X 0,Y 599.977,Z 1039.899,A -85,B 0,C 180,E1 28880.407,E2 28880.407} C_VEL
LIN {X 0,Y 600.131,Z 1033.43,A -85,B 0,C 180,E1 28877.979,E2 28877.979} C_VEL
LIN {X 0,Y 600.376,Z 1026.855,A -85,B 0,C 180,E1 28876.026,E2 28876.026} C_VEL
LIN {X 0,Y 600.809,Z 1017.709,A -85,B 0,C 180,E1 28873.764,E2 28873.764} C_VEL
LIN {X 0,Y 601.404,Z 1007.563,A -85,B 0,C 180,E1 28871.686,E2 28871.686} C_VEL
LIN {X 0,Y 602.235,Z 995.823,A -85,B 0,C 180,E1 28869.594,E2 28869.594} C_VEL
LIN {X 0,Y 603.299,Z 982.647,A -85,B 0,C 180,E1 28867.592,E2 28867.592} C_VEL
LIN {X 0,Y 604.779,Z 966.914,A -85,B 0,C 180,E1 28865.482,E2 28865.482} C_VEL
LIN {X 0,Y 606.352,Z 950.764,A -85,B 0,C 180,E1 28863.614,E2 28863.614} C_VEL
LIN {X 0,Y 608.209,Z 933.493,A -85,B 0,C 180,E1 28861.847,E2 28861.847} C_VEL
LIN {X 0,Y 610.106,Z 915.133,A -85,B 0,C 180,E1 28860.226,E2 28860.226} C_VEL
LIN {X 0,Y 612.122,Z 896.309,A -85,B 0,C 180,E1 28858.76,E2 28858.76} C_VEL
LIN {X 0,Y 614.194,Z 875.91,A -85,B 0,C 180,E1 28857.394,E2 28857.394} C_VEL
LIN {X 0,Y 615.954,Z 857.768,A -85,B 0,C 180,E1 28856.333,E2 28856.333} C_VEL
LIN {X 0,Y 617.994,Z 834.601,A -85,B 0,C 180,E1 28855.17,E2 28855.17} C_VEL
LIN {X 0,Y 619.641,Z 814.117,A -85,B 0,C 180,E1 28854.314,E2 28854.314} C_VEL
LIN {X 0,Y 621.335,Z 790.192,A -85,B 0,C 180,E1 28853.486,E2 28853.486} C_VEL
LIN {X 0,Y 622.573,Z 768.29,A -85,B 0,C 180,E1 28852.895,E2 28852.895} C_VEL
LIN {X 0,Y 623.558,Z 746.916,A -85,B 0,C 180,E1 28852.447,E2 28852.447} C_VEL
LIN {X 0,Y 624.385,Z 714.088,A -85,B 0,C 180,E1 28851.973,E2 28851.973} C_VEL
LIN {X 0,Y 629.115,Z 459.765,A -85,B 0,C 180,E1 28848.677,E2 28848.677} C_VEL
LIN {X 0,Y 630.263,Z 394.469,A -85,B 0,C 180,E1 28847.807,E2 28847.807} C_VEL
LIN {X 0,Y 616.493,Z 371.695,A -85,B 0,C 180,E1 28846.334,E2 28846.334} C_VEL
LIN {X 0,Y 604.629,Z 353.842,A -85,B 0,C 180,E1 28845.006,E2 28845.006} C_VEL
LIN {X 0,Y 602.702,Z 350.561,A -85,B 0,C 180,E1 28844.76,E2 28844.76} C_VEL
LIN {X 0,Y 601.12,Z 346.347,A -85,B 0,C 180,E1 28844.141,E2 28844.141} C_VEL
LIN {X 0,Y 601.072,Z 346.326,A -85,B 0,C 180,E1 28841.205,E2 28841.205} C_VEL
LIN {X 0,Y 601.127,Z 346.352,A -85,B 0,C 180,E1 28838.105,E2 28838.105} C_VEL
LIN {X 0,Y 601.077,Z 346.322,A -85,B 0,C 180,E1 28835.023,E2 28835.023} C_VEL
LIN {X 0,Y 601.104,Z 346.343,A -85,B 0,C 180,E1 28831.787,E2 28831.787} C_VEL
LIN {X 0,Y 601.084,Z 346.351,A -85,B 0,C 180,E1 28828.843,E2 28828.843} C_VEL
LIN {X 0,Y 601.088,Z 346.344,A -85,B 0,C 180,E1 28825.521,E2 28825.521} C_VEL
LIN {X 0,Y 601.096,Z 346.355,A -85,B 0,C 180,E1 28822.598,E2 28822.598} C_VEL
LIN {X 0,Y 601.083,Z 346.353,A -85,B 0,C 180,E1 28819.332,E2 28819.332} C_VEL
LIN {X 0,Y 601.113,Z 346.353,A -85,B 0,C 180,E1 28816.305,E2 28816.305} C_VEL
LIN {X 0,Y 601.078,Z 346.349,A -85,B 0,C 180,E1 28813.173,E2 28813.173} C_VEL
LIN {X 0,Y 601.116,Z 346.343,A -85,B 0,C 180,E1 28810.156,E2 28810.156} C_VEL
LIN {X 0,Y 601.076,Z 346.352,A -85,B 0,C 180,E1 28806.975,E2 28806.975} C_VEL
LIN {X 0,Y 601.13,Z 346.353,A -85,B 0,C 180,E1 28803.91,E2 28803.91} C_VEL
LIN {X 0,Y 601.071,Z 346.345,A -85,B 0,C 180,E1 28800.763,E2 28800.763} C_VEL
LIN {X 0,Y 601.135,Z 346.339,A -85,B 0,C 180,E1 28797.712,E2 28797.712} C_VEL
LIN {X 0,Y 601.072,Z 346.355,A -85,B 0,C 180,E1 28794.559,E2 28794.559} C_VEL
LIN {X 0,Y 601.14,Z 346.35,A -85,B 0,C 180,E1 28791.487,E2 28791.487} C_VEL
LIN {X 0,Y 601.071,Z 346.34,A -85,B 0,C 180,E1 28788.388,E2 28788.388} C_VEL
LIN {X 0,Y 601.132,Z 346.337,A -85,B 0,C 180,E1 28785.256,E2 28785.256} C_VEL
LIN {X 0,Y 601.076,Z 346.355,A -85,B 0,C 180,E1 28782.177,E2 28782.177} C_VEL
LIN {X 0,Y 601.107,Z 346.352,A -85,B 0,C 180,E1 28778.935,E2 28778.935} C_VEL
LIN {X 0,Y 601.074,Z 346.344,A -85,B 0,C 180,E1 28776.053,E2 28776.053} C_VEL
LIN {X 0,Y 601.108,Z 346.341,A -85,B 0,C 180,E1 28772.864,E2 28772.864} C_VEL
LIN {X 0,Y 601.078,Z 346.354,A -85,B 0,C 180,E1 28769.953,E2 28769.953} C_VEL
LIN {X 0,Y 601.103,Z 346.355,A -85,B 0,C 180,E1 28766.706,E2 28766.706} C_VEL
LIN {X 0,Y 601.079,Z 346.357,A -85,B 0,C 180,E1 28763.784,E2 28763.784} C_VEL
LIN {X 0,Y 601.093,Z 346.355,A -85,B 0,C 180,E1 28760.52,E2 28760.52} C_VEL
LIN {X 0,Y 601.079,Z 346.346,A -85,B 0,C 180,E1 28757.645,E2 28757.645} C_VEL
LIN {X 0,Y 601.088,Z 346.48,A -85,B 0,C 180,E1 28756.003,E2 28756.003} C_VEL
LIN {X 0,Y 602.408,Z 349.863,A -85,B 0,C 180,E1 28755.537,E2 28755.537} C_VEL
LIN {X 0,Y 610.096,Z 368.505,A -85,B 0,C 180,E1 28753.033,E2 28753.033} C_VEL
LIN {X 0,Y 612.618,Z 374.622,A -85,B 0,C 180,E1 28752.287,E2 28752.287} C_VEL
LIN {X 0,Y 626.907,Z 398.785,A -85,B 0,C 180,E1 28750.729,E2 28750.729} C_VEL
LIN {X 0,Y 630.302,Z 413.187,A -85,B 0,C 180,E1 28750.247,E2 28750.247} C_VEL
LIN {X 0,Y 625.305,Z 678.851,A -85,B 0,C 180,E1 28746.791,E2 28746.791} C_VEL
LIN {X 0,Y 623.609,Z 766.876,A -85,B 0,C 180,E1 28745.64,E2 28745.64} C_VEL
LIN {X 0,Y 622.513,Z 792.116,A -85,B 0,C 180,E1 28745.153,E2 28745.153} C_VEL
LIN {X 0,Y 621.327,Z 812.813,A -85,B 0,C 180,E1 28744.62,E2 28744.62} C_VEL
LIN {X 0,Y 619.815,Z 835.949,A -85,B 0,C 180,E1 28743.874,E2 28743.874} C_VEL
LIN {X 0,Y 618.029,Z 858.133,A -85,B 0,C 180,E1 28742.985,E2 28742.985} C_VEL
LIN {X 0,Y 616.219,Z 879.499,A -85,B 0,C 180,E1 28741.974,E2 28741.974} C_VEL
LIN {X 0,Y 614.165,Z 901.367,A -85,B 0,C 180,E1 28740.744,E2 28740.744} C_VEL
LIN {X 0,Y 612.36,Z 919.919,A -85,B 0,C 180,E1 28739.546,E2 28739.546} C_VEL
LIN {X 0,Y 610.169,Z 941.37,A -85,B 0,C 180,E1 28737.948,E2 28737.948} C_VEL
LIN {X 0,Y 608.466,Z 958.204,A -85,B 0,C 180,E1 28736.512,E2 28736.512} C_VEL
LIN {X 0,Y 606.561,Z 977.386,A -85,B 0,C 180,E1 28734.649,E2 28734.649} C_VEL
LIN {X 0,Y 605.093,Z 992.65,A -85,B 0,C 180,E1 28732.953,E2 28732.953} C_VEL
LIN {X 0,Y 603.751,Z 1007.707,A -85,B 0,C 180,E1 28731.062,E2 28731.062} C_VEL
LIN {X 0,Y 602.589,Z 1021.238,A -85,B 0,C 180,E1 28729.08,E2 28729.08} C_VEL
LIN {X 0,Y 601.668,Z 1033.688,A -85,B 0,C 180,E1 28727.007,E2 28727.007} C_VEL
LIN {X 0,Y 600.962,Z 1044.707,A -85,B 0,C 180,E1 28724.832,E2 28724.832} C_VEL
LIN {X 0,Y 600.515,Z 1053.583,A -85,B 0,C 180,E1 28722.794,E2 28722.794} C_VEL
LIN {X 0,Y 600.189,Z 1061.907,A -85,B 0,C 180,E1 28720.462,E2 28720.462} C_VEL
LIN {X 0,Y 600.028,Z 1067.491,A -85,B 0,C 180,E1 28718.529,E2 28718.529} C_VEL
LIN {X 0,Y 599.946,Z 1072.695,A -85,B 0,C 180,E1 28716.219,E2 28716.219} C_VEL
LIN {X 0,Y 599.911,Z 1076.009,A -85,B 0,C 180,E1 28714.014,E2 28714.014} C_VEL
LIN {X 0,Y 599.906,Z 1077.835,A -85,B 0,C 180,E1 28712.006,E2 28712.006} C_VEL
LIN {X 0,Y 599.895,Z 1078.417,A -85,B 0,C 180,E1 28709.618,E2 28709.618} C_VEL
LIN {X 0,Y 599.908,Z 1077.495,A -85,B 0,C 180,E1 28707.516,E2 28707.516} C_VEL
LIN {X 0,Y 599.925,Z 1075.085,A -85,B 0,C 180,E1 28705.22,E2 28705.22} C_VEL
LIN {X 0,Y 599.968,Z 1071.102,A -85,B 0,C 180,E1 28703.012,E2 28703.012} C_VEL
LIN {X 0,Y 600.05,Z 1066.219,A -85,B 0,C 180,E1 28700.988,E2 28700.988} C_VEL
LIN {X 0,Y 600.302,Z 1058.66,A -85,B 0,C 180,E1 28698.568,E2 28698.568} C_VEL
LIN {X 0,Y 600.649,Z 1050.747,A -85,B 0,C 180,E1 28696.523,E2 28696.523} C_VEL
LIN {X 0,Y 601.23,Z 1040.401,A -85,B 0,C 180,E1 28694.271,E2 28694.271} C_VEL
LIN {X 0,Y 601.991,Z 1029.111,A -85,B 0,C 180,E1 28692.205,E2 28692.205} C_VEL
LIN {X 0,Y 603.057,Z 1015.705,A -85,B 0,C 180,E1 28690.07,E2 28690.07} C_VEL
LIN {X 0,Y 604.209,Z 1002.366,A -85,B 0,C 180,E1 28688.242,E2 28688.242} C_VEL
LIN {X 0,Y 605.684,Z 986.675,A -85,B 0,C 180,E1 28686.35,E2 28686.35} C_VEL
LIN {X 0,Y 607.335,Z 969.481,A -85,B 0,C 180,E1 28684.552,E2 28684.552} C_VEL
LIN {X 0,Y 609.031,Z 952.779,A -85,B 0,C 180,E1 28683.003,E2 28683.003} C_VEL
LIN {X 0,Y 611.099,Z 932.382,A -85,B 0,C 180,E1 28681.353,E2 28681.353} C_VEL
LIN {X 0,Y 612.926,Z 914.014,A -85,B 0,C 180,E1 28680.054,E2 28680.054} C_VEL
LIN {X 0,Y 615.152,Z 891.169,A -85,B 0,C 180,E1 28678.658,E2 28678.658} C_VEL
LIN {X 0,Y 616.861,Z 872.159,A -85,B 0,C 180,E1 28677.662,E2 28677.662} C_VEL
LIN {X 0,Y 618.757,Z 849.985,A -85,B 0,C 180,E1 28676.664,E2 28676.664} C_VEL
LIN {X 0,Y 620.364,Z 827.239,A -85,B 0,C 180,E1 28675.826,E2 28675.826} C_VEL
LIN {X 0,Y 621.869,Z 804.051,A -85,B 0,C 180,E1 28675.131,E2 28675.131} C_VEL
LIN {X 0,Y 623.087,Z 780.045,A -85,B 0,C 180,E1 28674.594,E2 28674.594} C_VEL
LIN {X 0,Y 623.869,Z 757.754,A -85,B 0,C 180,E1 28674.229,E2 28674.229} C_VEL
LIN {X 0,Y 628.139,Z 514.362,A -85,B 0,C 180,E1 28671.097,E2 28671.097} C_VEL
LIN {X 0,Y 629.865,Z 412.184,A -85,B 0,C 180,E1 28669.757,E2 28669.757} C_VEL
LIN {X 0,Y 626.549,Z 398.688,A -85,B 0,C 180,E1 28669.309,E2 28669.309} C_VEL
LIN {X 0,Y 612.132,Z 374.17,A -85,B 0,C 180,E1 28667.798,E2 28667.798} C_VEL
LIN {X 0,Y 605.013,Z 356.379,A -85,B 0,C 180,E1 28665.558,E2 28665.558} C_VEL
LIN {X 0,Y 602.095,Z 349.342,A -85,B 0,C 180,E1 28664.626,E2 28664.626} C_VEL
LIN {X 0,Y 601.073,Z 346.362,A -85,B 0,C 180,E1 28664.218,E2 28664.218} C_VEL
LIN {X 0,Y 601.141,Z 346.354,A -85,B 0,C 180,E1 28661.107,E2 28661.107} C_VEL
LIN {X 0,Y 601.072,Z 346.354,A -85,B 0,C 180,E1 28657.988,E2 28657.988} C_VEL
LIN {X 0,Y 601.137,Z 346.344,A -85,B 0,C 180,E1 28654.903,E2 28654.903} C_VEL
LIN {X 0,Y 601.07,Z 346.351,A -85,B 0,C 180,E1 28651.826,E2 28651.826} C_VEL
LIN {X 0,Y 601.146,Z 346.349,A -85,B 0,C 180,E1 28648.731,E2 28648.731} C_VEL
LIN {X 0,Y 601.073,Z 346.353,A -85,B 0,C 180,E1 28645.627,E2 28645.627} C_VEL
LIN {X 0,Y 601.128,Z 346.34,A -85,B 0,C 180,E1 28642.493,E2 28642.493} C_VEL
LIN {X 0,Y 601.071,Z 346.344,A -85,B 0,C 180,E1 28639.534,E2 28639.534} C_VEL
LIN {X 0,Y 601.132,Z 346.354,A -85,B 0,C 180,E1 28636.426,E2 28636.426} C_VEL
LIN {X 0,Y 601.071,Z 346.348,A -85,B 0,C 180,E1 28633.467,E2 28633.467} C_VEL
LIN {X 0,Y 601.13,Z 346.339,A -85,B 0,C 180,E1 28630.349,E2 28630.349} C_VEL
LIN {X 0,Y 601.073,Z 346.354,A -85,B 0,C 180,E1 28627.359,E2 28627.359} C_VEL
LIN {X 0,Y 601.132,Z 346.334,A -85,B 0,C 180,E1 28624.293,E2 28624.293} C_VEL
LIN {X 0,Y 601.073,Z 346.353,A -85,B 0,C 180,E1 28621.237,E2 28621.237} C_VEL
LIN {X 0,Y 601.129,Z 346.339,A -85,B 0,C 180,E1 28618.094,E2 28618.094} C_VEL
LIN {X 0,Y 601.075,Z 346.346,A -85,B 0,C 180,E1 28615.038,E2 28615.038} C_VEL
LIN {X 0,Y 601.119,Z 346.354,A -85,B 0,C 180,E1 28611.872,E2 28611.872} C_VEL
LIN {X 0,Y 601.077,Z 346.335,A -85,B 0,C 180,E1 28608.874,E2 28608.874} C_VEL
LIN {X 0,Y 601.106,Z 346.351,A -85,B 0,C 180,E1 28605.65,E2 28605.65} C_VEL
LIN {X 0,Y 601.084,Z 346.347,A -85,B 0,C 180,E1 28602.677,E2 28602.677} C_VEL
LIN {X 0,Y 601.087,Z 346.339,A -85,B 0,C 180,E1 28599.35,E2 28599.35} C_VEL
LIN {X 0,Y 601.096,Z 346.353,A -85,B 0,C 180,E1 28596.428,E2 28596.428} C_VEL
LIN {X 0,Y 601.088,Z 346.357,A -85,B 0,C 180,E1 28593.205,E2 28593.205} C_VEL
LIN {X 0,Y 601.101,Z 346.337,A -85,B 0,C 180,E1 28590.263,E2 28590.263} C_VEL
LIN {X 0,Y 601.083,Z 346.343,A -85,B 0,C 180,E1 28587.046,E2 28587.046} C_VEL
LIN {X 0,Y 601.115,Z 346.351,A -85,B 0,C 180,E1 28584.043,E2 28584.043} C_VEL
LIN {X 0,Y 601.079,Z 346.351,A -85,B 0,C 180,E1 28580.822,E2 28580.822} C_VEL
LIN {X 0,Y 601.133,Z 346.345,A -85,B 0,C 180,E1 28577.779,E2 28577.779} C_VEL
LIN {X 0,Y 601.073,Z 346.328,A -85,B 0,C 180,E1 28574.603,E2 28574.603} C_VEL
LIN {X 0,Y 601.153,Z 346.432,A -85,B 0,C 180,E1 28571.513,E2 28571.513} C_VEL
LIN {X 0,Y 602.862,Z 351.065,A -85,B 0,C 180,E1 28570.924,E2 28570.924} C_VEL
LIN {X 0,Y 616.619,Z 372.529,A -85,B 0,C 180,E1 28569.441,E2 28569.441} C_VEL
LIN {X 0,Y 630.095,Z 394.837,A -85,B 0,C 180,E1 28568.059,E2 28568.059} C_VEL
LIN {X 0,Y 629.133,Z 447.61,A -85,B 0,C 180,E1 28567.368,E2 28567.368} C_VEL
LIN {X 0,Y 628.238,Z 455.306,A -85,B 0,C 180,E1 28567.323,E2 28567.323} C_VEL
LIN {X 0,Y 622.958,Z 475.869,A -85,B 0,C 180,E1 28567.417,E2 28567.417} C_VEL
LIN {X 0,Y 622.23,Z 482.476,A -85,B 0,C 180,E1 28567.376,E2 28567.376} C_VEL
LIN {X 0,Y 617.513,Z 731.123,A -85,B 0,C 180,E1 28564.143,E2 28564.143} C_VEL
LIN {X 0,Y 616.722,Z 753.294,A -85,B 0,C 180,E1 28563.773,E2 28563.773} C_VEL
LIN {X 0,Y 615.459,Z 777.86,A -85,B 0,C 180,E1 28563.208,E2 28563.208} C_VEL
LIN {X 0,Y 614.004,Z 799.911,A -85,B 0,C 180,E1 28562.534,E2 28562.534} C_VEL
LIN {X 0,Y 612.299,Z 822.879,A -85,B 0,C 180,E1 28561.675,E2 28561.675} C_VEL
LIN {X 0,Y 610.303,Z 844.777,A -85,B 0,C 180,E1 28560.668,E2 28560.668} C_VEL
LIN {X 0,Y 608.392,Z 864.519,A -85,B 0,C 180,E1 28559.609,E2 28559.609} C_VEL
LIN {X 0,Y 606.038,Z 886.679,A -85,B 0,C 180,E1 28558.214,E2 28558.214} C_VEL
LIN {X 0,Y 604.102,Z 904.459,A -85,B 0,C 180,E1 28556.923,E2 28556.923} C_VEL
LIN {X 0,Y 601.738,Z 925.356,A -85,B 0,C 180,E1 28555.175,E2 28555.175} C_VEL
LIN {X 0,Y 599.882,Z 941.946,A -85,B 0,C 180,E1 28553.58,E2 28553.58} C_VEL
LIN {X 0,Y 597.901,Z 960.025,A -85,B 0,C 180,E1 28551.587,E2 28551.587} C_VEL
LIN {X 0,Y 596.425,Z 974.226,A -85,B 0,C 180,E1 28549.794,E2 28549.794} C_VEL
LIN {X 0,Y 594.973,Z 989.307,A -85,B 0,C 180,E1 28547.608,E2 28547.608} C_VEL
LIN {X 0,Y 593.962,Z 1001.792,A -85,B 0,C 180,E1 28545.525,E2 28545.525} C_VEL
LIN {X 0,Y 593.142,Z 1013.486,A -85,B 0,C 180,E1 28543.254,E2 28543.254} C_VEL
LIN {X 0,Y 592.636,Z 1022.096,A -85,B 0,C 180,E1 28541.286,E2 28541.286} C_VEL
LIN {X 0,Y 592.261,Z 1030.49,A -85,B 0,C 180,E1 28539.018,E2 28539.018} C_VEL
LIN {X 0,Y 592.049,Z 1036.745,A -85,B 0,C 180,E1 28536.887,E2 28536.887} C_VEL
LIN {X 0,Y 591.963,Z 1041.511,A -85,B 0,C 180,E1 28534.845,E2 28534.845} C_VEL
LIN {X 0,Y 591.923,Z 1045.542,A -85,B 0,C 180,E1 28532.42,E2 28532.42} C_VEL
LIN {X 0,Y 591.905,Z 1047.554,A -85,B 0,C 180,E1 28530.387,E2 28530.387} C_VEL
LIN {X 0,Y 591.896,Z 1048.437,A -85,B 0,C 180,E1 28528.258,E2 28528.258} C_VEL
LIN {X 0,Y 591.913,Z 1047.773,A -85,B 0,C 180,E1 28525.834,E2 28525.834} C_VEL
LIN {X 0,Y 591.922,Z 1045.899,A -85,B 0,C 180,E1 28523.794,E2 28523.794} C_VEL
LIN {X 0,Y 591.95,Z 1042.329,A -85,B 0,C 180,E1 28521.452,E2 28521.452} C_VEL
LIN {X 0,Y 592.038,Z 1037.192,A -85,B 0,C 180,E1 28519.195,E2 28519.195} C_VEL
LIN {X 0,Y 592.239,Z 1031.206,A -85,B 0,C 180,E1 28517.123,E2 28517.123} C_VEL
LIN {X 0,Y 592.617,Z 1022.571,A -85,B 0,C 180,E1 28514.739,E2 28514.739} C_VEL
LIN {X 0,Y 593.118,Z 1013.869,A -85,B 0,C 180,E1 28512.74,E2 28512.74} C_VEL
LIN {X 0,Y 593.945,Z 1002.028,A -85,B 0,C 180,E1 28510.427,E2 28510.427} C_VEL
LIN {X 0,Y 594.974,Z 989.301,A -85,B 0,C 180,E1 28508.301,E2 28508.301} C_VEL
LIN {X 0,Y 596.458,Z 973.859,A -85,B 0,C 180,E1 28506.066,E2 28506.066} C_VEL
LIN {X 0,Y 597.891,Z 960.118,A -85,B 0,C 180,E1 28504.333,E2 28504.333} C_VEL
LIN {X 0,Y 599.873,Z 942.069,A -85,B 0,C 180,E1 28502.341,E2 28502.341} C_VEL
LIN {X 0,Y 601.647,Z 926.152,A -85,B 0,C 180,E1 28500.806,E2 28500.806} C_VEL
LIN {X 0,Y 603.862,Z 906.891,A -85,B 0,C 180,E1 28499.171,E2 28499.171} C_VEL
LIN {X 0,Y 605.902,Z 888.072,A -85,B 0,C 180,E1 28497.79,E2 28497.79} C_VEL
LIN {X 0,Y 608.117,Z 867.448,A -85,B 0,C 180,E1 28496.464,E2 28496.464} C_VEL
LIN {X 0,Y 610.217,Z 845.785,A -85,B 0,C 180,E1 28495.291,E2 28495.291} C_VEL
LIN {X 0,Y 612.113,Z 825.036,A -85,B 0,C 180,E1 28494.327,E2 28494.327} C_VEL
LIN {X 0,Y 613.912,Z 801.822,A -85,B 0,C 180,E1 28493.437,E2 28493.437} C_VEL
LIN {X 0,Y 615.308,Z 781.023,A -85,B 0,C 180,E1 28492.787,E2 28492.787} C_VEL
LIN {X 0,Y 616.707,Z 754.929,A -85,B 0,C 180,E1 28492.16,E2 28492.16} C_VEL
LIN {X 0,Y 617.54,Z 732.814,A -85,B 0,C 180,E1 28491.782,E2 28491.782} C_VEL
LIN {X 0,Y 622.504,Z 483.337,A -85,B 0,C 180,E1 28488.513,E2 28488.513} C_VEL
LIN {X 0,Y 624.172,Z 397.807,A -85,B 0,C 180,E1 28487.37,E2 28487.37} C_VEL
LIN {X 0,Y 611.713,Z 377.111,A -85,B 0,C 180,E1 28486.007,E2 28486.007} C_VEL
LIN {X 0,Y 600.335,Z 359.822,A -85,B 0,C 180,E1 28484.708,E2 28484.708} C_VEL
LIN {X 0,Y 594.515,Z 350.884,A -85,B 0,C 180,E1 28483.996,E2 28483.996} C_VEL
LIN {X 0,Y 593.137,Z 347.34,A -85,B 0,C 180,E1 28483.456,E2 28483.456} C_VEL
LIN {X 0,Y 593.201,Z 347.303,A -85,B 0,C 180,E1 28480.336,E2 28480.336} C_VEL
LIN {X 0,Y 593.135,Z 347.329,A -85,B 0,C 180,E1 28477.243,E2 28477.243} C_VEL
LIN {X 0,Y 593.186,Z 347.326,A -85,B 0,C 180,E1 28474.03,E2 28474.03} C_VEL
LIN {X 0,Y 593.138,Z 347.336,A -85,B 0,C 180,E1 28471.054,E2 28471.054} C_VEL
LIN {X 0,Y 593.191,Z 347.334,A -85,B 0,C 180,E1 28467.944,E2 28467.944} C_VEL
LIN {X 0,Y 593.139,Z 347.334,A -85,B 0,C 180,E1 28464.914,E2 28464.914} C_VEL
LIN {X 0,Y 593.169,Z 347.33,A -85,B 0,C 180,E1 28461.664,E2 28461.664} C_VEL
LIN {X 0,Y 593.146,Z 347.342,A -85,B 0,C 180,E1 28458.669,E2 28458.669} C_VEL
LIN {X 0,Y 593.148,Z 347.34,A -85,B 0,C 180,E1 28455.347,E2 28455.347} C_VEL
LIN {X 0,Y 593.152,Z 347.341,A -85,B 0,C 180,E1 28452.461,E2 28452.461} C_VEL
LIN {X 0,Y 593.14,Z 347.337,A -85,B 0,C 180,E1 28449.118,E2 28449.118} C_VEL
LIN {X 0,Y 593.166,Z 347.334,A -85,B 0,C 180,E1 28446.193,E2 28446.193} C_VEL
LIN {X 0,Y 593.139,Z 347.342,A -85,B 0,C 180,E1 28442.996,E2 28442.996} C_VEL
LIN {X 0,Y 593.177,Z 347.337,A -85,B 0,C 180,E1 28440,E2 28440} C_VEL
LIN {X 0,Y 593.135,Z 347.331,A -85,B 0,C 180,E1 28436.811,E2 28436.811} C_VEL
LIN {X 0,Y 593.195,Z 347.329,A -85,B 0,C 180,E1 28433.71,E2 28433.71} C_VEL
LIN {X 0,Y 593.134,Z 347.344,A -85,B 0,C 180,E1 28430.589,E2 28430.589} C_VEL
LIN {X 0,Y 593.199,Z 347.336,A -85,B 0,C 180,E1 28427.41,E2 28427.41} C_VEL
LIN {X 0,Y 593.131,Z 347.329,A -85,B 0,C 180,E1 28424.352,E2 28424.352} C_VEL
LIN {X 0,Y 593.191,Z 347.325,A -85,B 0,C 180,E1 28421.219,E2 28421.219} C_VEL
LIN {X 0,Y 593.135,Z 347.345,A -85,B 0,C 180,E1 28418.127,E2 28418.127} C_VEL
LIN {X 0,Y 593.178,Z 347.341,A -85,B 0,C 180,E1 28414.97,E2 28414.97} C_VEL
LIN {X 0,Y 593.139,Z 347.339,A -85,B 0,C 180,E1 28411.944,E2 28411.944} C_VEL
LIN {X 0,Y 593.16,Z 347.342,A -85,B 0,C 180,E1 28408.721,E2 28408.721} C_VEL
LIN {X 0,Y 593.146,Z 347.348,A -85,B 0,C 180,E1 28405.734,E2 28405.734} C_VEL
LIN {X 0,Y 593.142,Z 347.343,A -85,B 0,C 180,E1 28402.393,E2 28402.393} C_VEL
LIN {X 0,Y 593.157,Z 347.344,A -85,B 0,C 180,E1 28399.487,E2 28399.487} C_VEL
LIN {X 0,Y 593.203,Z 347.514,A -85,B 0,C 180,E1 28396.683,E2 28396.683} C_VEL
LIN {X 0,Y 594.313,Z 350.62,A -85,B 0,C 180,E1 28396.252,E2 28396.252} C_VEL
LIN {X 0,Y 599.743,Z 363.46,A -85,B 0,C 180,E1 28394.445,E2 28394.445} C_VEL
LIN {X 0,Y 604.178,Z 374.241,A -85,B 0,C 180,E1 28393.04,E2 28393.04} C_VEL
LIN {X 0,Y 615.048,Z 392.088,A -85,B 0,C 180,E1 28391.807,E2 28391.807} C_VEL
LIN {X 0,Y 621.799,Z 403.971,A -85,B 0,C 180,E1 28391.063,E2 28391.063} C_VEL
LIN {X 0,Y 624.187,Z 415.618,A -85,B 0,C 180,E1 28390.695,E2 28390.695} C_VEL
LIN {X 0,Y 618.894,Z 680.404,A -85,B 0,C 180,E1 28387.218,E2 28387.218} C_VEL
LIN {X 0,Y 617.125,Z 766.737,A -85,B 0,C 180,E1 28386.077,E2 28386.077} C_VEL
LIN {X 0,Y 615.96,Z 791.941,A -85,B 0,C 180,E1 28385.587,E2 28385.587} C_VEL
LIN {X 0,Y 614.692,Z 812.825,A -85,B 0,C 180,E1 28385.044,E2 28385.044} C_VEL
LIN {X 0,Y 612.984,Z 837.056,A -85,B 0,C 180,E1 28384.247,E2 28384.247} C_VEL
LIN {X 0,Y 611.217,Z 857.916,A -85,B 0,C 180,E1 28383.4,E2 28383.4} C_VEL
LIN {X 0,Y 609.321,Z 878.967,A -85,B 0,C 180,E1 28382.397,E2 28382.397} C_VEL
LIN {X 0,Y 607.109,Z 901.141,A -85,B 0,C 180,E1 28381.141,E2 28381.141} C_VEL
LIN {X 0,Y 605.152,Z 920.171,A -85,B 0,C 180,E1 28379.898,E2 28379.898} C_VEL
LIN {X 0,Y 602.881,Z 941.145,A -85,B 0,C 180,E1 28378.316,E2 28378.316} C_VEL
LIN {X 0,Y 601.038,Z 958.14,A -85,B 0,C 180,E1 28376.851,E2 28376.851} C_VEL
LIN {X 0,Y 599.032,Z 977.16,A -85,B 0,C 180,E1 28374.98,E2 28374.98} C_VEL
LIN {X 0,Y 597.458,Z 992.425,A -85,B 0,C 180,E1 28373.264,E2 28373.264} C_VEL
LIN {X 0,Y 595.961,Z 1008.237,A -85,B 0,C 180,E1 28371.248,E2 28371.248} C_VEL
LIN {X 0,Y 594.797,Z 1021.223,A -85,B 0,C 180,E1 28369.34,E2 28369.34} C_VEL
LIN {X 0,Y 593.816,Z 1033.688,A -85,B 0,C 180,E1 28367.239,E2 28367.239} C_VEL
LIN {X 0,Y 593.06,Z 1044.637,A -85,B 0,C 180,E1 28365.049,E2 28365.049} C_VEL
LIN {X 0,Y 592.57,Z 1053.582,A -85,B 0,C 180,E1 28362.969,E2 28362.969} C_VEL
LIN {X 0,Y 592.22,Z 1061.907,A -85,B 0,C 180,E1 28360.605,E2 28360.605} C_VEL
LIN {X 0,Y 592.033,Z 1067.745,A -85,B 0,C 180,E1 28358.547,E2 28358.547} C_VEL
LIN {X 0,Y 591.947,Z 1073.015,A -85,B 0,C 180,E1 28356.109,E2 28356.109} C_VEL
LIN {X 0,Y 591.912,Z 1076.008,A -85,B 0,C 180,E1 28354.068,E2 28354.068} C_VEL
LIN {X 0,Y 591.907,Z 1077.835,A -85,B 0,C 180,E1 28352.033,E2 28352.033} C_VEL
LIN {X 0,Y 591.895,Z 1078.417,A -85,B 0,C 180,E1 28349.613,E2 28349.613} C_VEL
LIN {X 0,Y 591.907,Z 1077.494,A -85,B 0,C 180,E1 28347.483,E2 28347.483} C_VEL
LIN {X 0,Y 591.928,Z 1075.085,A -85,B 0,C 180,E1 28345.155,E2 28345.155} C_VEL
LIN {X 0,Y 591.98,Z 1071.102,A -85,B 0,C 180,E1 28342.917,E2 28342.917} C_VEL
LIN {X 0,Y 592.069,Z 1066.219,A -85,B 0,C 180,E1 28340.866,E2 28340.866} C_VEL
LIN {X 0,Y 592.341,Z 1058.659,A -85,B 0,C 180,E1 28338.412,E2 28338.412} C_VEL
LIN {X 0,Y 592.713,Z 1050.747,A -85,B 0,C 180,E1 28336.339,E2 28336.339} C_VEL
LIN {X 0,Y 593.342,Z 1040.4,A -85,B 0,C 180,E1 28334.057,E2 28334.057} C_VEL
LIN {X 0,Y 594.115,Z 1029.683,A -85,B 0,C 180,E1 28332.062,E2 28332.062} C_VEL
LIN {X 0,Y 595.078,Z 1018.012,A -85,B 0,C 180,E1 28330.159,E2 28330.159} C_VEL
LIN {X 0,Y 596.44,Z 1002.925,A -85,B 0,C 180,E1 28328.047,E2 28328.047} C_VEL
LIN {X 0,Y 597.812,Z 989.017,A -85,B 0,C 180,E1 28326.333,E2 28326.333} C_VEL
LIN {X 0,Y 599.748,Z 970.285,A -85,B 0,C 180,E1 28324.312,E2 28324.312} C_VEL
LIN {X 0,Y 601.538,Z 953.68,A -85,B 0,C 180,E1 28322.746,E2 28322.746} C_VEL
LIN {X 0,Y 603.791,Z 932.835,A -85,B 0,C 180,E1 28321.028,E2 28321.028} C_VEL
LIN {X 0,Y 605.723,Z 914.534,A -85,B 0,C 180,E1 28319.715,E2 28319.715} C_VEL
LIN {X 0,Y 608.081,Z 891.856,A -85,B 0,C 180,E1 28318.307,E2 28318.307} C_VEL
LIN {X 0,Y 609.97,Z 871.941,A -85,B 0,C 180,E1 28317.252,E2 28317.252} C_VEL
LIN {X 0,Y 611.957,Z 849.956,A -85,B 0,C 180,E1 28316.253,E2 28316.253} C_VEL
LIN {X 0,Y 613.666,Z 826.975,A -85,B 0,C 180,E1 28315.401,E2 28315.401} C_VEL
LIN {X 0,Y 615.272,Z 803.625,A -85,B 0,C 180,E1 28314.698,E2 28314.698} C_VEL
LIN {X 0,Y 616.529,Z 779.786,A -85,B 0,C 180,E1 28314.164,E2 28314.164} C_VEL
LIN {X 0,Y 617.343,Z 757.549,A -85,B 0,C 180,E1 28313.797,E2 28313.797} C_VEL
LIN {X 0,Y 621.875,Z 513.243,A -85,B 0,C 180,E1 28310.626,E2 28310.626} C_VEL
LIN {X 0,Y 623.645,Z 413.984,A -85,B 0,C 180,E1 28309.311,E2 28309.311} C_VEL
LIN {X 0,Y 620.948,Z 402.893,A -85,B 0,C 180,E1 28308.939,E2 28308.939} C_VEL
LIN {X 0,Y 606.513,Z 378.526,A -85,B 0,C 180,E1 28307.4,E2 28307.4} C_VEL
LIN {X 0,Y 603.652,Z 373.695,A -85,B 0,C 180,E1 28307.066,E2 28307.066} C_VEL
LIN {X 0,Y 596.249,Z 354.957,A -85,B 0,C 180,E1 28304.64,E2 28304.64} C_VEL
LIN {X 0,Y 593.174,Z 347.515,A -85,B 0,C 180,E1 28303.62,E2 28303.62} C_VEL
LIN {X 0,Y 593.143,Z 347.338,A -85,B 0,C 180,E1 28300.341,E2 28300.341} C_VEL
LIN {X 0,Y 593.154,Z 347.335,A -85,B 0,C 180,E1 28297.442,E2 28297.442} C_VEL
LIN {X 0,Y 593.137,Z 347.335,A -85,B 0,C 180,E1 28294.136,E2 28294.136} C_VEL
LIN {X 0,Y 593.179,Z 347.329,A -85,B 0,C 180,E1 28291.095,E2 28291.095} C_VEL
LIN {X 0,Y 593.135,Z 347.333,A -85,B 0,C 180,E1 28287.946,E2 28287.946} C_VEL
LIN {X 0,Y 593.198,Z 347.34,A -85,B 0,C 180,E1 28284.817,E2 28284.817} C_VEL
LIN {X 0,Y 593.132,Z 347.344,A -85,B 0,C 180,E1 28281.741,E2 28281.741} C_VEL
LIN {X 0,Y 593.196,Z 347.323,A -85,B 0,C 180,E1 28278.679,E2 28278.679} C_VEL
LIN {X 0,Y 593.133,Z 347.338,A -85,B 0,C 180,E1 28275.548,E2 28275.548} C_VEL
LIN {X 0,Y 593.199,Z 347.337,A -85,B 0,C 180,E1 28272.46,E2 28272.46} C_VEL
LIN {X 0,Y 593.134,Z 347.325,A -85,B 0,C 180,E1 28269.313,E2 28269.313} C_VEL
LIN {X 0,Y 593.176,Z 347.337,A -85,B 0,C 180,E1 28266.096,E2 28266.096} C_VEL
LIN {X 0,Y 593.139,Z 347.337,A -85,B 0,C 180,E1 28263.092,E2 28263.092} C_VEL
LIN {X 0,Y 593.156,Z 347.324,A -85,B 0,C 180,E1 28259.807,E2 28259.807} C_VEL
LIN {X 0,Y 593.152,Z 347.341,A -85,B 0,C 180,E1 28256.811,E2 28256.811} C_VEL
LIN {X 0,Y 593.142,Z 347.33,A -85,B 0,C 180,E1 28253.515,E2 28253.515} C_VEL
LIN {X 0,Y 593.174,Z 347.34,A -85,B 0,C 180,E1 28250.491,E2 28250.491} C_VEL
LIN {X 0,Y 593.138,Z 347.343,A -85,B 0,C 180,E1 28247.242,E2 28247.242} C_VEL
LIN {X 0,Y 593.189,Z 347.326,A -85,B 0,C 180,E1 28244.253,E2 28244.253} C_VEL
LIN {X 0,Y 593.138,Z 347.343,A -85,B 0,C 180,E1 28241.115,E2 28241.115} C_VEL
LIN {X 0,Y 593.203,Z 347.327,A -85,B 0,C 180,E1 28237.982,E2 28237.982} C_VEL
LIN {X 0,Y 593.136,Z 347.327,A -85,B 0,C 180,E1 28234.858,E2 28234.858} C_VEL
LIN {X 0,Y 593.203,Z 347.335,A -85,B 0,C 180,E1 28231.728,E2 28231.728} C_VEL
LIN {X 0,Y 593.138,Z 347.344,A -85,B 0,C 180,E1 28228.72,E2 28228.72} C_VEL
LIN {X 0,Y 593.196,Z 347.333,A -85,B 0,C 180,E1 28225.62,E2 28225.62} C_VEL
LIN {X 0,Y 593.139,Z 347.342,A -85,B 0,C 180,E1 28222.514,E2 28222.514} C_VEL
LIN {X 0,Y 593.184,Z 347.337,A -85,B 0,C 180,E1 28219.335,E2 28219.335} C_VEL
LIN {X 0,Y 593.142,Z 347.303,A -85,B 0,C 180,E1 28216.278,E2 28216.278} C_VEL
LIN {X 0,Y 593.154,Z 347.344,A -85,B 0,C 180,E1 28212.924,E2 28212.924} C_VEL
LIN {X 0,Y 593.154,Z 347.392,A -85,B 0,C 180,E1 28212.161,E2 28212.161} C_VEL
LIN {X 0,Y 594.654,Z 351.038,A -85,B 0,C 180,E1 28211.651,E2 28211.651} C_VEL
LIN {X 0,Y 597.659,Z 355.727,A -85,B 0,C 180,E1 28211.307,E2 28211.307} C_VEL
LIN {X 0,Y 614.201,Z 381.749,A -85,B 0,C 180,E1 28209.497,E2 28209.497} C_VEL
LIN {X 0,Y 623.877,Z 398.119,A -85,B 0,C 180,E1 28208.486,E2 28208.486} C_VEL
LIN {X 0,Y 622.23,Z 482.476,A -85,B 0,C 180,E1 28207.376,E2 28207.376} C_VEL
LIN {X 0,Y 621.294,Z 490.172,A -85,B 0,C 180,E1 28207.333,E2 28207.333} C_VEL
LIN {X 0,Y 616.011,Z 510.726,A -85,B 0,C 180,E1 28207.429,E2 28207.429} C_VEL
LIN {X 0,Y 615.282,Z 517.33,A -85,B 0,C 180,E1 28207.387,E2 28207.387} C_VEL
LIN {X 0,Y 610.798,Z 738.818,A -85,B 0,C 180,E1 28204.47,E2 28204.47} C_VEL
LIN {X 0,Y 609.666,Z 764.83,A -85,B 0,C 180,E1 28203.966,E2 28203.966} C_VEL
LIN {X 0,Y 608.431,Z 785.229,A -85,B 0,C 180,E1 28203.432,E2 28203.432} C_VEL
LIN {X 0,Y 606.832,Z 808.119,A -85,B 0,C 180,E1 28202.684,E2 28202.684} C_VEL
LIN {X 0,Y 604.856,Z 830.468,A -85,B 0,C 180,E1 28201.77,E2 28201.77} C_VEL
LIN {X 0,Y 602.904,Z 851.104,A -85,B 0,C 180,E1 28200.773,E2 28200.773} C_VEL
LIN {X 0,Y 600.587,Z 872.854,A -85,B 0,C 180,E1 28199.525,E2 28199.525} C_VEL
LIN {X 0,Y 598.536,Z 891.142,A -85,B 0,C 180,E1 28198.311,E2 28198.311} C_VEL
LIN {X 0,Y 596.051,Z 912.338,A -85,B 0,C 180,E1 28196.687,E2 28196.687} C_VEL
LIN {X 0,Y 594.016,Z 929.15,A -85,B 0,C 180,E1 28195.206,E2 28195.206} C_VEL
LIN {X 0,Y 591.899,Z 947.25,A -85,B 0,C 180,E1 28193.39,E2 28193.39} C_VEL
LIN {X 0,Y 590.061,Z 962.964,A -85,B 0,C 180,E1 28191.575,E2 28191.575} C_VEL
LIN {X 0,Y 588.41,Z 978.342,A -85,B 0,C 180,E1 28189.558,E2 28189.558} C_VEL
LIN {X 0,Y 587.046,Z 991.568,A -85,B 0,C 180,E1 28187.546,E2 28187.546} C_VEL
LIN {X 0,Y 585.976,Z 1003.957,A -85,B 0,C 180,E1 28185.398,E2 28185.398} C_VEL
LIN {X 0,Y 585.111,Z 1015.437,A -85,B 0,C 180,E1 28183.037,E2 28183.037} C_VEL
LIN {X 0,Y 584.562,Z 1024.976,A -85,B 0,C 180,E1 28180.745,E2 28180.745} C_VEL
LIN {X 0,Y 584.217,Z 1032.642,A -85,B 0,C 180,E1 28178.464,E2 28178.464} C_VEL
LIN {X 0,Y 584.029,Z 1038.844,A -85,B 0,C 180,E1 28176.192,E2 28176.192} C_VEL
LIN {X 0,Y 583.939,Z 1043.53,A -85,B 0,C 180,E1 28173.829,E2 28173.829} C_VEL
LIN {X 0,Y 583.916,Z 1046.369,A -85,B 0,C 180,E1 28171.766,E2 28171.766} C_VEL
LIN {X 0,Y 583.905,Z 1048.193,A -85,B 0,C 180,E1 28169.313,E2 28169.313} C_VEL
LIN {X 0,Y 583.901,Z 1048.322,A -85,B 0,C 180,E1 28167.153,E2 28167.153} C_VEL
LIN {X 0,Y 583.907,Z 1047.208,A -85,B 0,C 180,E1 28164.99,E2 28164.99} C_VEL
LIN {X 0,Y 583.921,Z 1044.246,A -85,B 0,C 180,E1 28162.522,E2 28162.522} C_VEL
LIN {X 0,Y 583.981,Z 1040.488,A -85,B 0,C 180,E1 28160.481,E2 28160.481} C_VEL
LIN {X 0,Y 584.138,Z 1034.778,A -85,B 0,C 180,E1 28158.147,E2 28158.147} C_VEL
LIN {X 0,Y 584.42,Z 1027.715,A -85,B 0,C 180,E1 28155.939,E2 28155.939} C_VEL
LIN {X 0,Y 584.85,Z 1019.591,A -85,B 0,C 180,E1 28153.819,E2 28153.819} C_VEL
LIN {X 0,Y 585.612,Z 1008.323,A -85,B 0,C 180,E1 28151.38,E2 28151.38} C_VEL
LIN {X 0,Y 586.517,Z 997.396,A -85,B 0,C 180,E1 28149.336,E2 28149.336} C_VEL
LIN {X 0,Y 587.799,Z 983.988,A -85,B 0,C 180,E1 28147.18,E2 28147.18} C_VEL
LIN {X 0,Y 589.206,Z 970.769,A -85,B 0,C 180,E1 28145.325,E2 28145.325} C_VEL
LIN {X 0,Y 591.158,Z 953.447,A -85,B 0,C 180,E1 28143.207,E2 28143.207} C_VEL
LIN {X 0,Y 592.998,Z 937.922,A -85,B 0,C 180,E1 28141.553,E2 28141.553} C_VEL
LIN {X 0,Y 595.316,Z 918.528,A -85,B 0,C 180,E1 28139.743,E2 28139.743} C_VEL
LIN {X 0,Y 597.342,Z 901.341,A -85,B 0,C 180,E1 28138.347,E2 28138.347} C_VEL
LIN {X 0,Y 599.727,Z 881.124,A -85,B 0,C 180,E1 28136.906,E2 28136.906} C_VEL
LIN {X 0,Y 601.926,Z 860.711,A -85,B 0,C 180,E1 28135.664,E2 28135.664} C_VEL
LIN {X 0,Y 604.066,Z 839.682,A -85,B 0,C 180,E1 28134.554,E2 28134.554} C_VEL
LIN {X 0,Y 606.1,Z 817.103,A -85,B 0,C 180,E1 28133.566,E2 28133.566} C_VEL
LIN {X 0,Y 607.771,Z 795.967,A -85,B 0,C 180,E1 28132.794,E2 28132.794} C_VEL
LIN {X 0,Y 609.435,Z 771.119,A -85,B 0,C 180,E1 28132.079,E2 28132.079} C_VEL
LIN {X 0,Y 610.501,Z 750.521,A -85,B 0,C 180,E1 28131.627,E2 28131.627} C_VEL
LIN {X 0,Y 611.38,Z 724.593,A -85,B 0,C 180,E1 28131.214,E2 28131.214} C_VEL
LIN {X 0,Y 616.675,Z 471.092,A -85,B 0,C 180,E1 28127.868,E2 28127.868} C_VEL
LIN {X 0,Y 618.093,Z 401.034,A -85,B 0,C 180,E1 28126.92,E2 28126.92} C_VEL
LIN {X 0,Y 606.633,Z 382.039,A -85,B 0,C 180,E1 28125.638,E2 28125.638} C_VEL
LIN {X 0,Y 596.058,Z 365.802,A -85,B 0,C 180,E1 28124.406,E2 28124.406} C_VEL
LIN {X 0,Y 589.397,Z 356.043,A -85,B 0,C 180,E1 28123.6,E2 28123.6} C_VEL
LIN {X 0,Y 586.094,Z 351.126,A -85,B 0,C 180,E1 28123.166,E2 28123.166} C_VEL
LIN {X 0,Y 585.241,Z 348.333,A -85,B 0,C 180,E1 28122.722,E2 28122.722} C_VEL
LIN {X 0,Y 585.198,Z 348.309,A -85,B 0,C 180,E1 28119.593,E2 28119.593} C_VEL
LIN {X 0,Y 585.238,Z 348.294,A -85,B 0,C 180,E1 28116.582,E2 28116.582} C_VEL
LIN {X 0,Y 585.198,Z 348.333,A -85,B 0,C 180,E1 28113.38,E2 28113.38} C_VEL
LIN {X 0,Y 585.268,Z 348.331,A -85,B 0,C 180,E1 28110.178,E2 28110.178} C_VEL
LIN {X 0,Y 585.199,Z 348.333,A -85,B 0,C 180,E1 28107.033,E2 28107.033} C_VEL
LIN {X 0,Y 585.239,Z 348.331,A -85,B 0,C 180,E1 28103.779,E2 28103.779} C_VEL
LIN {X 0,Y 585.201,Z 348.325,A -85,B 0,C 180,E1 28100.818,E2 28100.818} C_VEL
LIN {X 0,Y 585.225,Z 348.321,A -85,B 0,C 180,E1 28097.565,E2 28097.565} C_VEL
LIN {X 0,Y 585.208,Z 348.326,A -85,B 0,C 180,E1 28094.547,E2 28094.547} C_VEL
LIN {X 0,Y 585.207,Z 348.329,A -85,B 0,C 180,E1 28091.232,E2 28091.232} C_VEL
LIN {X 0,Y 585.236,Z 348.33,A -85,B 0,C 180,E1 28088.153,E2 28088.153} C_VEL
LIN {X 0,Y 585.199,Z 348.324,A -85,B 0,C 180,E1 28084.999,E2 28084.999} C_VEL
LIN {X 0,Y 585.252,Z 348.316,A -85,B 0,C 180,E1 28081.86,E2 28081.86} C_VEL
LIN {X 0,Y 585.195,Z 348.333,A -85,B 0,C 180,E1 28078.727,E2 28078.727} C_VEL
LIN {X 0,Y 585.258,Z 348.329,A -85,B 0,C 180,E1 28075.591,E2 28075.591} C_VEL
LIN {X 0,Y 585.192,Z 348.317,A -85,B 0,C 180,E1 28072.539,E2 28072.539} C_VEL
LIN {X 0,Y 585.251,Z 348.315,A -85,B 0,C 180,E1 28069.367,E2 28069.367} C_VEL
LIN {X 0,Y 585.197,Z 348.334,A -85,B 0,C 180,E1 28066.261,E2 28066.261} C_VEL
LIN {X 0,Y 585.229,Z 348.33,A -85,B 0,C 180,E1 28063.013,E2 28063.013} C_VEL
LIN {X 0,Y 585.203,Z 348.318,A -85,B 0,C 180,E1 28060.008,E2 28060.008} C_VEL
LIN {X 0,Y 585.204,Z 348.317,A -85,B 0,C 180,E1 28056.647,E2 28056.647} C_VEL
LIN {X 0,Y 585.229,Z 348.323,A -85,B 0,C 180,E1 28053.626,E2 28053.626} C_VEL
LIN {X 0,Y 585.2,Z 348.331,A -85,B 0,C 180,E1 28050.41,E2 28050.41} C_VEL
LIN {X 0,Y 585.249,Z 348.331,A -85,B 0,C 180,E1 28047.324,E2 28047.324} C_VEL
LIN {X 0,Y 585.194,Z 348.336,A -85,B 0,C 180,E1 28044.121,E2 28044.121} C_VEL
LIN {X 0,Y 585.26,Z 348.328,A -85,B 0,C 180,E1 28040.919,E2 28040.919} C_VEL
LIN {X 0,Y 585.194,Z 348.326,A -85,B 0,C 180,E1 28037.864,E2 28037.864} C_VEL
LIN {X 0,Y 585.223,Z 348.344,A -85,B 0,C 180,E1 28037.422,E2 28037.422} C_VEL
LIN {X 0,Y 586.681,Z 351.97,A -85,B 0,C 180,E1 28036.887,E2 28036.887} C_VEL
LIN {X 0,Y 593.473,Z 368.351,A -85,B 0,C 180,E1 28034.547,E2 28034.547} C_VEL
LIN {X 0,Y 595.931,Z 373.949,A -85,B 0,C 180,E1 28033.805,E2 28033.805} C_VEL
LIN {X 0,Y 609.554,Z 396.18,A -85,B 0,C 180,E1 28032.215,E2 28032.215} C_VEL
LIN {X 0,Y 616.287,Z 408.139,A -85,B 0,C 180,E1 28031.455,E2 28031.455} C_VEL
LIN {X 0,Y 618.126,Z 417.453,A -85,B 0,C 180,E1 28031.16,E2 28031.16} C_VEL
LIN {X 0,Y 612.536,Z 681.518,A -85,B 0,C 180,E1 28027.661,E2 28027.661} C_VEL
LIN {X 0,Y 610.689,Z 766.523,A -85,B 0,C 180,E1 28026.526,E2 28026.526} C_VEL
LIN {X 0,Y 609.446,Z 791.914,A -85,B 0,C 180,E1 28026.029,E2 28026.029} C_VEL
LIN {X 0,Y 608.087,Z 813.136,A -85,B 0,C 180,E1 28025.471,E2 28025.471} C_VEL
LIN {X 0,Y 606.241,Z 837.672,A -85,B 0,C 180,E1 28024.65,E2 28024.65} C_VEL
LIN {X 0,Y 604.447,Z 857.777,A -85,B 0,C 180,E1 28023.824,E2 28023.824} C_VEL
LIN {X 0,Y 602.438,Z 878.777,A -85,B 0,C 180,E1 28022.813,E2 28022.813} C_VEL
LIN {X 0,Y 600.086,Z 900.917,A -85,B 0,C 180,E1 28021.547,E2 28021.547} C_VEL
LIN {X 0,Y 597.986,Z 920.207,A -85,B 0,C 180,E1 28020.274,E2 28020.274} C_VEL
LIN {X 0,Y 595.62,Z 940.919,A -85,B 0,C 180,E1 28018.693,E2 28018.693} C_VEL
LIN {X 0,Y 593.657,Z 957.901,A -85,B 0,C 180,E1 28017.213,E2 28017.213} C_VEL
LIN {X 0,Y 591.447,Z 977.584,A -85,B 0,C 180,E1 28015.248,E2 28015.248} C_VEL
LIN {X 0,Y 589.845,Z 992.199,A -85,B 0,C 180,E1 28013.582,E2 28013.582} C_VEL
LIN {X 0,Y 588.248,Z 1008.013,A -85,B 0,C 180,E1 28011.54,E2 28011.54} C_VEL
LIN {X 0,Y 586.994,Z 1020.999,A -85,B 0,C 180,E1 28009.607,E2 28009.607} C_VEL
LIN {X 0,Y 585.964,Z 1033.662,A -85,B 0,C 180,E1 28007.468,E2 28007.468} C_VEL
LIN {X 0,Y 585.19,Z 1044.177,A -85,B 0,C 180,E1 28005.358,E2 28005.358} C_VEL
LIN {X 0,Y 584.663,Z 1052.897,A -85,B 0,C 180,E1 28003.317,E2 28003.317} C_VEL
LIN {X 0,Y 584.256,Z 1061.604,A -85,B 0,C 180,E1 28000.851,E2 28000.851} C_VEL
LIN {X 0,Y 584.044,Z 1067.491,A -85,B 0,C 180,E1 27998.764,E2 27998.764} C_VEL
LIN {X 0,Y 583.946,Z 1072.695,A -85,B 0,C 180,E1 27996.39,E2 27996.39} C_VEL
LIN {X 0,Y 583.915,Z 1075.894,A -85,B 0,C 180,E1 27994.223,E2 27994.223} C_VEL
LIN {X 0,Y 583.909,Z 1077.766,A -85,B 0,C 180,E1 27992.159,E2 27992.159} C_VEL
LIN {X 0,Y 583.898,Z 1078.439,A -85,B 0,C 180,E1 27989.706,E2 27989.706} C_VEL
LIN {X 0,Y 583.908,Z 1077.562,A -85,B 0,C 180,E1 27987.546,E2 27987.546} C_VEL
LIN {X 0,Y 583.922,Z 1075.439,A -85,B 0,C 180,E1 27985.384,E2 27985.384} C_VEL
LIN {X 0,Y 583.982,Z 1071.308,A -85,B 0,C 180,E1 27982.919,E2 27982.919} C_VEL
LIN {X 0,Y 584.077,Z 1066.474,A -85,B 0,C 180,E1 27980.839,E2 27980.839} C_VEL
LIN {X 0,Y 584.348,Z 1059.365,A -85,B 0,C 180,E1 27978.451,E2 27978.451} C_VEL
LIN {X 0,Y 584.735,Z 1051.556,A -85,B 0,C 180,E1 27976.351,E2 27976.351} C_VEL
LIN {X 0,Y 585.357,Z 1041.888,A -85,B 0,C 180,E1 27974.139,E2 27974.139} C_VEL
LIN {X 0,Y 586.229,Z 1030.138,A -85,B 0,C 180,E1 27971.915,E2 27971.915} C_VEL
LIN {X 0,Y 587.241,Z 1018.436,A -85,B 0,C 180,E1 27969.987,E2 27969.987} C_VEL
LIN {X 0,Y 588.68,Z 1003.484,A -85,B 0,C 180,E1 27967.848,E2 27967.848} C_VEL
LIN {X 0,Y 590.127,Z 989.651,A -85,B 0,C 180,E1 27966.112,E2 27966.112} C_VEL
LIN {X 0,Y 592.068,Z 972.111,A -85,B 0,C 180,E1 27964.169,E2 27964.169} C_VEL
LIN {X 0,Y 593.989,Z 955.14,A -85,B 0,C 180,E1 27962.533,E2 27962.533} C_VEL
LIN {X 0,Y 596.231,Z 935.921,A -85,B 0,C 180,E1 27960.895,E2 27960.895} C_VEL
LIN {X 0,Y 598.376,Z 916.536,A -85,B 0,C 180,E1 27959.47,E2 27959.47} C_VEL
LIN {X 0,Y 600.66,Z 896.054,A -85,B 0,C 180,E1 27958.15,E2 27958.15} C_VEL
LIN {X 0,Y 602.819,Z 874.727,A -85,B 0,C 180,E1 27956.984,E2 27956.984} C_VEL
LIN {X 0,Y 604.633,Z 855.575,A -85,B 0,C 180,E1 27956.083,E2 27956.083} C_VEL
LIN {X 0,Y 606.634,Z 831.946,A -85,B 0,C 180,E1 27955.147,E2 27955.147} C_VEL
LIN {X 0,Y 608.207,Z 809.82,A -85,B 0,C 180,E1 27954.445,E2 27954.445} C_VEL
LIN {X 0,Y 609.71,Z 785.451,A -85,B 0,C 180,E1 27953.838,E2 27953.838} C_VEL
LIN {X 0,Y 610.708,Z 761.524,A -85,B 0,C 180,E1 27953.419,E2 27953.419} C_VEL
LIN {X 0,Y 615.333,Z 527.23,A -85,B 0,C 180,E1 27950.344,E2 27950.344} C_VEL
LIN {X 0,Y 617.477,Z 415.813,A -85,B 0,C 180,E1 27948.859,E2 27948.859} C_VEL
LIN {X 0,Y 615.289,Z 406.929,A -85,B 0,C 180,E1 27948.553,E2 27948.553} C_VEL
LIN {X 0,Y 601.355,Z 383.428,A -85,B 0,C 180,E1 27947.039,E2 27947.039} C_VEL
LIN {X 0,Y 595.404,Z 373.516,A -85,B 0,C 180,E1 27946.353,E2 27946.353} C_VEL
LIN {X 0,Y 588.035,Z 355.483,A -85,B 0,C 180,E1 27943.929,E2 27943.929} C_VEL
LIN {X 0,Y 585.253,Z 348.332,A -85,B 0,C 180,E1 27942.902,E2 27942.902} C_VEL
LIN {X 0,Y 585.194,Z 348.325,A -85,B 0,C 180,E1 27939.847,E2 27939.847} C_VEL
LIN {X 0,Y 585.246,Z 348.322,A -85,B 0,C 180,E1 27936.725,E2 27936.725} C_VEL
LIN {X 0,Y 585.201,Z 348.327,A -85,B 0,C 180,E1 27933.614,E2 27933.614} C_VEL
LIN {X 0,Y 585.212,Z 348.324,A -85,B 0,C 180,E1 27930.267,E2 27930.267} C_VEL
LIN {X 0,Y 585.209,Z 348.316,A -85,B 0,C 180,E1 27927.362,E2 27927.362} C_VEL
LIN {X 0,Y 585.206,Z 348.32,A -85,B 0,C 180,E1 27924.102,E2 27924.102} C_VEL
LIN {X 0,Y 585.211,Z 348.331,A -85,B 0,C 180,E1 27921.237,E2 27921.237} C_VEL
LIN {X 0,Y 585.202,Z 348.33,A -85,B 0,C 180,E1 27917.88,E2 27917.88} C_VEL
LIN {X 0,Y 585.251,Z 348.314,A -85,B 0,C 180,E1 27914.761,E2 27914.761} C_VEL
LIN {X 0,Y 585.197,Z 348.332,A -85,B 0,C 180,E1 27911.632,E2 27911.632} C_VEL
LIN {X 0,Y 585.262,Z 348.313,A -85,B 0,C 180,E1 27908.432,E2 27908.432} C_VEL
LIN {X 0,Y 585.195,Z 348.322,A -85,B 0,C 180,E1 27905.392,E2 27905.392} C_VEL
LIN {X 0,Y 585.25,Z 348.331,A -85,B 0,C 180,E1 27902.154,E2 27902.154} C_VEL
LIN {X 0,Y 585.196,Z 348.31,A -85,B 0,C 180,E1 27899.119,E2 27899.119} C_VEL
LIN {X 0,Y 585.233,Z 348.328,A -85,B 0,C 180,E1 27895.885,E2 27895.885} C_VEL
LIN {X 0,Y 585.206,Z 348.322,A -85,B 0,C 180,E1 27892.835,E2 27892.835} C_VEL
LIN {X 0,Y 585.204,Z 348.314,A -85,B 0,C 180,E1 27889.466,E2 27889.466} C_VEL
LIN {X 0,Y 585.242,Z 348.329,A -85,B 0,C 180,E1 27886.363,E2 27886.363} C_VEL
LIN {X 0,Y 585.199,Z 348.322,A -85,B 0,C 180,E1 27883.216,E2 27883.216} C_VEL
LIN {X 0,Y 585.256,Z 348.321,A -85,B 0,C 180,E1 27880.124,E2 27880.124} C_VEL
LIN {X 0,Y 585.2,Z 348.333,A -85,B 0,C 180,E1 27876.966,E2 27876.966} C_VEL
LIN {X 0,Y 585.259,Z 348.313,A -85,B 0,C 180,E1 27873.846,E2 27873.846} C_VEL
LIN {X 0,Y 585.198,Z 348.318,A -85,B 0,C 180,E1 27870.747,E2 27870.747} C_VEL
LIN {X 0,Y 585.252,Z 348.321,A -85,B 0,C 180,E1 27867.557,E2 27867.557} C_VEL
LIN {X 0,Y 585.207,Z 348.332,A -85,B 0,C 180,E1 27864.419,E2 27864.419} C_VEL
LIN {X 0,Y 585.213,Z 348.33,A -85,B 0,C 180,E1 27861.041,E2 27861.041} C_VEL
LIN {X 0,Y 585.23,Z 348.332,A -85,B 0,C 180,E1 27858.006,E2 27858.006} C_VEL
LIN {X 0,Y 585.199,Z 348.297,A -85,B 0,C 180,E1 27854.745,E2 27854.745} C_VEL
LIN {X 0,Y 585.229,Z 348.482,A -85,B 0,C 180,E1 27852.812,E2 27852.812} C_VEL
LIN {X 0,Y 586.433,Z 351.703,A -85,B 0,C 180,E1 27852.396,E2 27852.396} C_VEL
LIN {X 0,Y 593.873,Z 362.855,A -85,B 0,C 180,E1 27851.53,E2 27851.53} C_VEL
LIN {X 0,Y 604.368,Z 379.261,A -85,B 0,C 180,E1 27850.352,E2 27850.352} C_VEL
LIN {X 0,Y 617.684,Z 401.085,A -85,B 0,C 180,E1 27848.927,E2 27848.927} C_VEL
LIN {X 0,Y 615.282,Z 517.33,A -85,B 0,C 180,E1 27847.387,E2 27847.387} C_VEL
LIN {X 0,Y 614.34,Z 525.026,A -85,B 0,C 180,E1 27847.344,E2 27847.344} C_VEL
LIN {X 0,Y 609.054,Z 545.579,A -85,B 0,C 180,E1 27847.441,E2 27847.441} C_VEL
LIN {X 0,Y 608.331,Z 552.182,A -85,B 0,C 180,E1 27847.398,E2 27847.398} C_VEL
LIN {X 0,Y 604.333,Z 739.177,A -85,B 0,C 180,E1 27844.913,E2 27844.913} C_VEL
LIN {X 0,Y 603.148,Z 765.149,A -85,B 0,C 180,E1 27844.405,E2 27844.405} C_VEL
LIN {X 0,Y 601.853,Z 785.645,A -85,B 0,C 180,E1 27843.864,E2 27843.864} C_VEL
LIN {X 0,Y 600.119,Z 809.127,A -85,B 0,C 180,E1 27843.085,E2 27843.085} C_VEL
LIN {X 0,Y 598.083,Z 831.195,A -85,B 0,C 180,E1 27842.173,E2 27842.173} C_VEL
LIN {X 0,Y 596.041,Z 851.797,A -85,B 0,C 180,E1 27841.166,E2 27841.166} C_VEL
LIN {X 0,Y 593.605,Z 873.488,A -85,B 0,C 180,E1 27839.907,E2 27839.907} C_VEL
LIN {X 0,Y 591.43,Z 891.995,A -85,B 0,C 180,E1 27838.665,E2 27838.665} C_VEL
LIN {X 0,Y 588.808,Z 913.18,A -85,B 0,C 180,E1 27837.016,E2 27837.016} C_VEL
LIN {X 0,Y 586.698,Z 929.682,A -85,B 0,C 180,E1 27835.542,E2 27835.542} C_VEL
LIN {X 0,Y 584.333,Z 948.637,A -85,B 0,C 180,E1 27833.604,E2 27833.604} C_VEL
LIN {X 0,Y 582.508,Z 963.422,A -85,B 0,C 180,E1 27831.869,E2 27831.869} C_VEL
LIN {X 0,Y 580.746,Z 978.759,A -85,B 0,C 180,E1 27829.827,E2 27829.827} C_VEL
LIN {X 0,Y 579.359,Z 991.345,A -85,B 0,C 180,E1 27827.891,E2 27827.891} C_VEL
LIN {X 0,Y 578.223,Z 1003.569,A -85,B 0,C 180,E1 27825.753,E2 27825.753} C_VEL
LIN {X 0,Y 577.31,Z 1014.368,A -85,B 0,C 180,E1 27823.522,E2 27823.522} C_VEL
LIN {X 0,Y 576.729,Z 1022.773,A -85,B 0,C 180,E1 27821.501,E2 27821.501} C_VEL
LIN {X 0,Y 576.277,Z 1031.524,A -85,B 0,C 180,E1 27818.984,E2 27818.984} C_VEL
LIN {X 0,Y 576.058,Z 1037.458,A -85,B 0,C 180,E1 27816.855,E2 27816.855} C_VEL
LIN {X 0,Y 575.954,Z 1042.62,A -85,B 0,C 180,E1 27814.481,E2 27814.481} C_VEL
LIN {X 0,Y 575.921,Z 1045.947,A -85,B 0,C 180,E1 27812.189,E2 27812.189} C_VEL
LIN {X 0,Y 575.923,Z 1047.796,A -85,B 0,C 180,E1 27810.099,E2 27810.099} C_VEL
LIN {X 0,Y 575.895,Z 1048.429,A -85,B 0,C 180,E1 27807.612,E2 27807.612} C_VEL
LIN {X 0,Y 575.904,Z 1047.597,A -85,B 0,C 180,E1 27805.519,E2 27805.519} C_VEL
LIN {X 0,Y 575.925,Z 1045.605,A -85,B 0,C 180,E1 27803.42,E2 27803.42} C_VEL
LIN {X 0,Y 575.978,Z 1041.588,A -85,B 0,C 180,E1 27800.911,E2 27800.911} C_VEL
LIN {X 0,Y 576.085,Z 1036.789,A -85,B 0,C 180,E1 27798.791,E2 27798.791} C_VEL
LIN {X 0,Y 576.351,Z 1030.1,A -85,B 0,C 180,E1 27796.455,E2 27796.455} C_VEL
LIN {X 0,Y 576.806,Z 1021.575,A -85,B 0,C 180,E1 27794.104,E2 27794.104} C_VEL
LIN {X 0,Y 577.502,Z 1011.945,A -85,B 0,C 180,E1 27791.841,E2 27791.841} C_VEL
LIN {X 0,Y 578.438,Z 1000.88,A -85,B 0,C 180,E1 27789.669,E2 27789.669} C_VEL
LIN {X 0,Y 579.584,Z 989.371,A -85,B 0,C 180,E1 27787.695,E2 27787.695} C_VEL
LIN {X 0,Y 581.192,Z 974.619,A -85,B 0,C 180,E1 27785.505,E2 27785.505} C_VEL
LIN {X 0,Y 582.82,Z 960.91,A -85,B 0,C 180,E1 27783.728,E2 27783.728} C_VEL
LIN {X 0,Y 584.986,Z 943.44,A -85,B 0,C 180,E1 27781.741,E2 27781.741} C_VEL
LIN {X 0,Y 587.079,Z 926.87,A -85,B 0,C 180,E1 27780.102,E2 27780.102} C_VEL
LIN {X 0,Y 589.511,Z 907.89,A -85,B 0,C 180,E1 27778.449,E2 27778.449} C_VEL
LIN {X 0,Y 591.868,Z 888.411,A -85,B 0,C 180,E1 27776.987,E2 27776.987} C_VEL
LIN {X 0,Y 594.357,Z 867.821,A -85,B 0,C 180,E1 27775.638,E2 27775.638} C_VEL
LIN {X 0,Y 596.576,Z 847.233,A -85,B 0,C 180,E1 27774.497,E2 27774.497} C_VEL
LIN {X 0,Y 598.546,Z 827.813,A -85,B 0,C 180,E1 27773.568,E2 27773.568} C_VEL
LIN {X 0,Y 600.712,Z 803.148,A -85,B 0,C 180,E1 27772.588,E2 27772.588} C_VEL
LIN {X 0,Y 602.28,Z 782.045,A -85,B 0,C 180,E1 27771.913,E2 27771.913} C_VEL
LIN {X 0,Y 603.8,Z 756.854,A -85,B 0,C 180,E1 27771.289,E2 27771.289} C_VEL
LIN {X 0,Y 604.744,Z 734.357,A -85,B 0,C 180,E1 27770.893,E2 27770.893} C_VEL
LIN {X 0,Y 610.261,Z 487.129,A -85,B 0,C 180,E1 27767.59,E2 27767.59} C_VEL
LIN {X 0,Y 612.064,Z 404.383,A -85,B 0,C 180,E1 27766.463,E2 27766.463} C_VEL
LIN {X 0,Y 601.821,Z 387.309,A -85,B 0,C 180,E1 27765.291,E2 27765.291} C_VEL
LIN {X 0,Y 591.561,Z 371.457,A -85,B 0,C 180,E1 27764.071,E2 27764.071} C_VEL
LIN {X 0,Y 584.635,Z 361.326,A -85,B 0,C 180,E1 27763.217,E2 27763.217} C_VEL
LIN {X 0,Y 577.839,Z 351.31,A -85,B 0,C 180,E1 27762.309,E2 27762.309} C_VEL
LIN {X 0,Y 577.29,Z 349.299,A -85,B 0,C 180,E1 27762.009,E2 27762.009} C_VEL
LIN {X 0,Y 577.273,Z 349.313,A -85,B 0,C 180,E1 27758.949,E2 27758.949} C_VEL
LIN {X 0,Y 577.263,Z 349.277,A -85,B 0,C 180,E1 27755.591,E2 27755.591} C_VEL
LIN {X 0,Y 577.31,Z 349.315,A -85,B 0,C 180,E1 27752.474,E2 27752.474} C_VEL
LIN {X 0,Y 577.262,Z 349.321,A -85,B 0,C 180,E1 27749.353,E2 27749.353} C_VEL
LIN {X 0,Y 577.313,Z 349.316,A -85,B 0,C 180,E1 27746.32,E2 27746.32} C_VEL
LIN {X 0,Y 577.259,Z 349.323,A -85,B 0,C 180,E1 27743.108,E2 27743.108} C_VEL
LIN {X 0,Y 577.322,Z 349.319,A -85,B 0,C 180,E1 27739.95,E2 27739.95} C_VEL
LIN {X 0,Y 577.259,Z 349.317,A -85,B 0,C 180,E1 27736.814,E2 27736.814} C_VEL
LIN {X 0,Y 577.301,Z 349.308,A -85,B 0,C 180,E1 27733.624,E2 27733.624} C_VEL
LIN {X 0,Y 577.263,Z 349.316,A -85,B 0,C 180,E1 27730.58,E2 27730.58} C_VEL
LIN {X 0,Y 577.275,Z 349.318,A -85,B 0,C 180,E1 27727.264,E2 27727.264} C_VEL
LIN {X 0,Y 577.277,Z 349.316,A -85,B 0,C 180,E1 27724.271,E2 27724.271} C_VEL
LIN {X 0,Y 577.263,Z 349.31,A -85,B 0,C 180,E1 27720.992,E2 27720.992} C_VEL
LIN {X 0,Y 577.299,Z 349.31,A -85,B 0,C 180,E1 27717.97,E2 27717.97} C_VEL
LIN {X 0,Y 577.258,Z 349.322,A -85,B 0,C 180,E1 27714.733,E2 27714.733} C_VEL
LIN {X 0,Y 577.323,Z 349.311,A -85,B 0,C 180,E1 27711.635,E2 27711.635} C_VEL
LIN {X 0,Y 577.255,Z 349.305,A -85,B 0,C 180,E1 27708.409,E2 27708.409} C_VEL
LIN {X 0,Y 577.312,Z 349.303,A -85,B 0,C 180,E1 27705.25,E2 27705.25} C_VEL
LIN {X 0,Y 577.262,Z 349.322,A -85,B 0,C 180,E1 27702.146,E2 27702.146} C_VEL
LIN {X 0,Y 577.273,Z 349.32,A -85,B 0,C 180,E1 27698.776,E2 27698.776} C_VEL
LIN {X 0,Y 577.269,Z 349.31,A -85,B 0,C 180,E1 27695.872,E2 27695.872} C_VEL
LIN {X 0,Y 577.267,Z 349.311,A -85,B 0,C 180,E1 27692.565,E2 27692.565} C_VEL
LIN {X 0,Y 577.285,Z 349.322,A -85,B 0,C 180,E1 27689.606,E2 27689.606} C_VEL
LIN {X 0,Y 577.261,Z 349.324,A -85,B 0,C 180,E1 27686.339,E2 27686.339} C_VEL
LIN {X 0,Y 577.319,Z 349.32,A -85,B 0,C 180,E1 27683.146,E2 27683.146} C_VEL
LIN {X 0,Y 577.256,Z 349.327,A -85,B 0,C 180,E1 27680.012,E2 27680.012} C_VEL
LIN {X 0,Y 577.26,Z 349.335,A -85,B 0,C 180,E1 27678.174,E2 27678.174} C_VEL
LIN {X 0,Y 578.661,Z 352.927,A -85,B 0,C 180,E1 27677.631,E2 27677.631} C_VEL
LIN {X 0,Y 585.725,Z 369.544,A -85,B 0,C 180,E1 27675.168,E2 27675.168} C_VEL
LIN {X 0,Y 587.445,Z 373.637,A -85,B 0,C 180,E1 27674.627,E2 27674.627} C_VEL
LIN {X 0,Y 598.918,Z 391.689,A -85,B 0,C 180,E1 27673.237,E2 27673.237} C_VEL
LIN {X 0,Y 610.774,Z 412.128,A -85,B 0,C 180,E1 27671.86,E2 27671.86} C_VEL
LIN {X 0,Y 612.108,Z 419.351,A -85,B 0,C 180,E1 27671.634,E2 27671.634} C_VEL
LIN {X 0,Y 606.224,Z 682.374,A -85,B 0,C 180,E1 27668.117,E2 27668.117} C_VEL
LIN {X 0,Y 604.297,Z 766.416,A -85,B 0,C 180,E1 27666.984,E2 27666.984} C_VEL
LIN {X 0,Y 602.985,Z 791.763,A -85,B 0,C 180,E1 27666.484,E2 27666.484} C_VEL
LIN {X 0,Y 601.544,Z 813.171,A -85,B 0,C 180,E1 27665.916,E2 27665.916} C_VEL
LIN {X 0,Y 599.667,Z 836.921,A -85,B 0,C 180,E1 27665.118,E2 27665.118} C_VEL
LIN {X 0,Y 597.684,Z 858.052,A -85,B 0,C 180,E1 27664.242,E2 27664.242} C_VEL
LIN {X 0,Y 595.5,Z 879.666,A -85,B 0,C 180,E1 27663.187,E2 27663.187} C_VEL
LIN {X 0,Y 593.014,Z 901.561,A -85,B 0,C 180,E1 27661.911,E2 27661.911} C_VEL
LIN {X 0,Y 590.645,Z 922.212,A -85,B 0,C 180,E1 27660.522,E2 27660.522} C_VEL
LIN {X 0,Y 588.151,Z 942.533,A -85,B 0,C 180,E1 27658.925,E2 27658.925} C_VEL
LIN {X 0,Y 585.978,Z 960.488,A -85,B 0,C 180,E1 27657.323,E2 27657.323} C_VEL
LIN {X 0,Y 583.805,Z 978.579,A -85,B 0,C 180,E1 27655.461,E2 27655.461} C_VEL
LIN {X 0,Y 582.063,Z 993.683,A -85,B 0,C 180,E1 27653.702,E2 27653.702} C_VEL
LIN {X 0,Y 580.309,Z 1009.914,A -85,B 0,C 180,E1 27651.531,E2 27651.531} C_VEL
LIN {X 0,Y 579.089,Z 1022.06,A -85,B 0,C 180,E1 27649.676,E2 27649.676} C_VEL
LIN {X 0,Y 577.919,Z 1035.491,A -85,B 0,C 180,E1 27647.313,E2 27647.313} C_VEL
LIN {X 0,Y 577.186,Z 1045.421,A -85,B 0,C 180,E1 27645.267,E2 27645.267} C_VEL
LIN {X 0,Y 576.602,Z 1055.128,A -85,B 0,C 180,E1 27642.926,E2 27642.926} C_VEL
LIN {X 0,Y 576.249,Z 1062.512,A -85,B 0,C 180,E1 27640.7,E2 27640.7} C_VEL
LIN {X 0,Y 576.044,Z 1068.762,A -85,B 0,C 180,E1 27638.384,E2 27638.384} C_VEL
LIN {X 0,Y 575.946,Z 1073.493,A -85,B 0,C 180,E1 27635.979,E2 27635.979} C_VEL
LIN {X 0,Y 575.91,Z 1076.235,A -85,B 0,C 180,E1 27633.982,E2 27633.982} C_VEL
LIN {X 0,Y 575.895,Z 1078.104,A -85,B 0,C 180,E1 27631.691,E2 27631.691} C_VEL
LIN {X 0,Y 575.895,Z 1078.371,A -85,B 0,C 180,E1 27629.403,E2 27629.403} C_VEL
LIN {X 0,Y 575.907,Z 1077.425,A -85,B 0,C 180,E1 27627.313,E2 27627.313} C_VEL
LIN {X 0,Y 575.932,Z 1074.929,A -85,B 0,C 180,E1 27624.92,E2 27624.92} C_VEL
LIN {X 0,Y 575.984,Z 1070.895,A -85,B 0,C 180,E1 27622.619,E2 27622.619} C_VEL
LIN {X 0,Y 576.125,Z 1065.965,A -85,B 0,C 180,E1 27620.51,E2 27620.51} C_VEL
LIN {X 0,Y 576.434,Z 1058.305,A -85,B 0,C 180,E1 27617.986,E2 27617.986} C_VEL
LIN {X 0,Y 576.827,Z 1051.101,A -85,B 0,C 180,E1 27616.058,E2 27616.058} C_VEL
LIN {X 0,Y 577.499,Z 1041.233,A -85,B 0,C 180,E1 27613.814,E2 27613.814} C_VEL
LIN {X 0,Y 578.433,Z 1029.338,A -85,B 0,C 180,E1 27611.558,E2 27611.558} C_VEL
LIN {X 0,Y 579.681,Z 1016.287,A -85,B 0,C 180,E1 27609.398,E2 27609.398} C_VEL
LIN {X 0,Y 581.178,Z 1001.706,A -85,B 0,C 180,E1 27607.333,E2 27607.333} C_VEL
LIN {X 0,Y 582.858,Z 986.869,A -85,B 0,C 180,E1 27605.471,E2 27605.471} C_VEL
LIN {X 0,Y 584.909,Z 969.334,A -85,B 0,C 180,E1 27603.556,E2 27603.556} C_VEL
LIN {X 0,Y 586.941,Z 952.681,A -85,B 0,C 180,E1 27601.954,E2 27601.954} C_VEL
LIN {X 0,Y 589.459,Z 931.724,A -85,B 0,C 180,E1 27600.198,E2 27600.198} C_VEL
LIN {X 0,Y 591.662,Z 913.344,A -85,B 0,C 180,E1 27598.86,E2 27598.86} C_VEL
LIN {X 0,Y 594.275,Z 890.446,A -85,B 0,C 180,E1 27597.424,E2 27597.424} C_VEL
LIN {X 0,Y 596.269,Z 871.373,A -85,B 0,C 180,E1 27596.401,E2 27596.401} C_VEL
LIN {X 0,Y 598.459,Z 849.276,A -85,B 0,C 180,E1 27595.385,E2 27595.385} C_VEL
LIN {X 0,Y 600.34,Z 826.581,A -85,B 0,C 180,E1 27594.533,E2 27594.533} C_VEL
LIN {X 0,Y 602.136,Z 802.945,A -85,B 0,C 180,E1 27593.815,E2 27593.815} C_VEL
LIN {X 0,Y 603.49,Z 779.272,A -85,B 0,C 180,E1 27593.279,E2 27593.279} C_VEL
LIN {X 0,Y 604.371,Z 757.158,A -85,B 0,C 180,E1 27592.909,E2 27592.909} C_VEL
LIN {X 0,Y 609.472,Z 510.586,A -85,B 0,C 180,E1 27589.651,E2 27589.651} C_VEL
LIN {X 0,Y 611.336,Z 417.63,A -85,B 0,C 180,E1 27588.398,E2 27588.398} C_VEL
LIN {X 0,Y 609.66,Z 410.943,A -85,B 0,C 180,E1 27588.16,E2 27588.16} C_VEL
LIN {X 0,Y 594.048,Z 384.607,A -85,B 0,C 180,E1 27586.419,E2 27586.419} C_VEL
LIN {X 0,Y 586.872,Z 372.967,A -85,B 0,C 180,E1 27585.551,E2 27585.551} C_VEL
LIN {X 0,Y 581.128,Z 359.046,A -85,B 0,C 180,E1 27583.627,E2 27583.627} C_VEL
LIN {X 0,Y 578.336,Z 352.395,A -85,B 0,C 180,E1 27582.667,E2 27582.667} C_VEL
LIN {X 0,Y 577.259,Z 349.329,A -85,B 0,C 180,E1 27582.227,E2 27582.227} C_VEL
LIN {X 0,Y 577.306,Z 349.313,A -85,B 0,C 180,E1 27579.211,E2 27579.211} C_VEL
LIN {X 0,Y 577.257,Z 349.326,A -85,B 0,C 180,E1 27576.011,E2 27576.011} C_VEL
LIN {X 0,Y 577.321,Z 349.316,A -85,B 0,C 180,E1 27572.827,E2 27572.827} C_VEL
LIN {X 0,Y 577.257,Z 349.32,A -85,B 0,C 180,E1 27569.696,E2 27569.696} C_VEL
LIN {X 0,Y 577.307,Z 349.305,A -85,B 0,C 180,E1 27566.542,E2 27566.542} C_VEL
LIN {X 0,Y 577.259,Z 349.304,A -85,B 0,C 180,E1 27563.478,E2 27563.478} C_VEL
LIN {X 0,Y 577.289,Z 349.313,A -85,B 0,C 180,E1 27560.268,E2 27560.268} C_VEL
LIN {X 0,Y 577.27,Z 349.318,A -85,B 0,C 180,E1 27557.229,E2 27557.229} C_VEL
LIN {X 0,Y 577.263,Z 349.309,A -85,B 0,C 180,E1 27553.83,E2 27553.83} C_VEL
LIN {X 0,Y 577.299,Z 349.315,A -85,B 0,C 180,E1 27550.781,E2 27550.781} C_VEL
LIN {X 0,Y 577.257,Z 349.323,A -85,B 0,C 180,E1 27547.565,E2 27547.565} C_VEL
LIN {X 0,Y 577.314,Z 349.298,A -85,B 0,C 180,E1 27544.47,E2 27544.47} C_VEL
LIN {X 0,Y 577.256,Z 349.32,A -85,B 0,C 180,E1 27541.29,E2 27541.29} C_VEL
LIN {X 0,Y 577.313,Z 349.302,A -85,B 0,C 180,E1 27538.114,E2 27538.114} C_VEL
LIN {X 0,Y 577.26,Z 349.313,A -85,B 0,C 180,E1 27535.032,E2 27535.032} C_VEL
LIN {X 0,Y 577.287,Z 349.324,A -85,B 0,C 180,E1 27531.734,E2 27531.734} C_VEL
LIN {X 0,Y 577.277,Z 349.297,A -85,B 0,C 180,E1 27528.625,E2 27528.625} C_VEL
LIN {X 0,Y 577.265,Z 349.316,A -85,B 0,C 180,E1 27525.351,E2 27525.351} C_VEL
LIN {X 0,Y 577.306,Z 349.311,A -85,B 0,C 180,E1 27522.252,E2 27522.252} C_VEL
LIN {X 0,Y 577.259,Z 349.304,A -85,B 0,C 180,E1 27519.095,E2 27519.095} C_VEL
LIN {X 0,Y 577.322,Z 349.314,A -85,B 0,C 180,E1 27515.983,E2 27515.983} C_VEL
LIN {X 0,Y 577.261,Z 349.322,A -85,B 0,C 180,E1 27512.788,E2 27512.788} C_VEL
LIN {X 0,Y 577.316,Z 349.306,A -85,B 0,C 180,E1 27509.6,E2 27509.6} C_VEL
LIN {X 0,Y 577.266,Z 349.307,A -85,B 0,C 180,E1 27506.458,E2 27506.458} C_VEL
LIN {X 0,Y 577.279,Z 349.31,A -85,B 0,C 180,E1 27503.151,E2 27503.151} C_VEL
LIN {X 0,Y 577.282,Z 349.311,A -85,B 0,C 180,E1 27500.112,E2 27500.112} C_VEL
LIN {X 0,Y 577.263,Z 349.286,A -85,B 0,C 180,E1 27496.821,E2 27496.821} C_VEL
LIN {X 0,Y 577.319,Z 349.314,A -85,B 0,C 180,E1 27493.617,E2 27493.617} C_VEL
LIN {X 0,Y 577.364,Z 349.61,A -85,B 0,C 180,E1 27493.478,E2 27493.478} C_VEL
LIN {X 0,Y 578.083,Z 351.909,A -85,B 0,C 180,E1 27493.192,E2 27493.192} C_VEL
LIN {X 0,Y 589.065,Z 368.125,A -85,B 0,C 180,E1 27491.881,E2 27491.881} C_VEL
LIN {X 0,Y 599.651,Z 384.804,A -85,B 0,C 180,E1 27490.669,E2 27490.669} C_VEL
LIN {X 0,Y 611.538,Z 404.499,A -85,B 0,C 180,E1 27489.368,E2 27489.368} C_VEL
LIN {X 0,Y 608.331,Z 552.182,A -85,B 0,C 180,E1 27487.398,E2 27487.398} C_VEL
LIN {X 0,Y 607.39,Z 559.879,A -85,B 0,C 180,E1 27487.355,E2 27487.355} C_VEL
LIN {X 0,Y 602.071,Z 580.427,A -85,B 0,C 180,E1 27487.455,E2 27487.455} C_VEL
LIN {X 0,Y 601.344,Z 587.031,A -85,B 0,C 180,E1 27487.412,E2 27487.412} C_VEL
LIN {X 0,Y 597.896,Z 739.693,A -85,B 0,C 180,E1 27485.364,E2 27485.364} C_VEL
LIN {X 0,Y 596.657,Z 765.553,A -85,B 0,C 180,E1 27484.852,E2 27484.852} C_VEL
LIN {X 0,Y 595.299,Z 786.138,A -85,B 0,C 180,E1 27484.303,E2 27484.303} C_VEL
LIN {X 0,Y 593.462,Z 809.785,A -85,B 0,C 180,E1 27483.509,E2 27483.509} C_VEL
LIN {X 0,Y 591.452,Z 830.775,A -85,B 0,C 180,E1 27482.635,E2 27482.635} C_VEL
LIN {X 0,Y 589.403,Z 850.476,A -85,B 0,C 180,E1 27481.672,E2 27481.672} C_VEL
LIN {X 0,Y 586.743,Z 873.279,A -85,B 0,C 180,E1 27480.35,E2 27480.35} C_VEL
LIN {X 0,Y 584.411,Z 892.18,A -85,B 0,C 180,E1 27479.072,E2 27479.072} C_VEL
LIN {X 0,Y 581.704,Z 913.116,A -85,B 0,C 180,E1 27477.43,E2 27477.43} C_VEL
LIN {X 0,Y 579.405,Z 930.214,A -85,B 0,C 180,E1 27475.888,E2 27475.888} C_VEL
LIN {X 0,Y 576.902,Z 949.117,A -85,B 0,C 180,E1 27473.927,E2 27473.927} C_VEL
LIN {X 0,Y 574.971,Z 963.88,A -85,B 0,C 180,E1 27472.171,E2 27472.171} C_VEL
LIN {X 0,Y 573.009,Z 979.861,A -85,B 0,C 180,E1 27470,E2 27470} C_VEL
LIN {X 0,Y 571.557,Z 992.364,A -85,B 0,C 180,E1 27468.038,E2 27468.038} C_VEL
LIN {X 0,Y 570.304,Z 1004.995,A -85,B 0,C 180,E1 27465.769,E2 27465.769} C_VEL
LIN {X 0,Y 569.362,Z 1015.611,A -85,B 0,C 180,E1 27463.507,E2 27463.507} C_VEL
LIN {X 0,Y 568.703,Z 1025.057,A -85,B 0,C 180,E1 27461.151,E2 27461.151} C_VEL
LIN {X 0,Y 568.28,Z 1032.626,A -85,B 0,C 180,E1 27458.805,E2 27458.805} C_VEL
LIN {X 0,Y 568.051,Z 1038.751,A -85,B 0,C 180,E1 27456.468,E2 27456.468} C_VEL
LIN {X 0,Y 567.949,Z 1043.461,A -85,B 0,C 180,E1 27454.038,E2 27454.038} C_VEL
LIN {X 0,Y 567.919,Z 1046.319,A -85,B 0,C 180,E1 27451.917,E2 27451.917} C_VEL
LIN {X 0,Y 567.901,Z 1048.16,A -85,B 0,C 180,E1 27449.496,E2 27449.496} C_VEL
LIN {X 0,Y 567.897,Z 1048.354,A -85,B 0,C 180,E1 27447.275,E2 27447.275} C_VEL
LIN {X 0,Y 567.9,Z 1047.431,A -85,B 0,C 180,E1 27445.239,E2 27445.239} C_VEL
LIN {X 0,Y 567.933,Z 1044.955,A -85,B 0,C 180,E1 27442.819,E2 27442.819} C_VEL
LIN {X 0,Y 567.988,Z 1040.906,A -85,B 0,C 180,E1 27440.475,E2 27440.475} C_VEL
LIN {X 0,Y 568.157,Z 1035.504,A -85,B 0,C 180,E1 27438.117,E2 27438.117} C_VEL
LIN {X 0,Y 568.499,Z 1028.326,A -85,B 0,C 180,E1 27435.724,E2 27435.724} C_VEL
LIN {X 0,Y 568.971,Z 1020.772,A -85,B 0,C 180,E1 27433.643,E2 27433.643} C_VEL
LIN {X 0,Y 569.837,Z 1010.002,A -85,B 0,C 180,E1 27431.164,E2 27431.164} C_VEL
LIN {X 0,Y 570.781,Z 999.79,A -85,B 0,C 180,E1 27429.169,E2 27429.169} C_VEL
LIN {X 0,Y 572.206,Z 986.821,A -85,B 0,C 180,E1 27426.957,E2 27426.957} C_VEL
LIN {X 0,Y 573.828,Z 973.072,A -85,B 0,C 180,E1 27424.949,E2 27424.949} C_VEL
LIN {X 0,Y 575.83,Z 957.495,A -85,B 0,C 180,E1 27422.939,E2 27422.939} C_VEL
LIN {X 0,Y 578.075,Z 940.311,A -85,B 0,C 180,E1 27421.033,E2 27421.033} C_VEL
LIN {X 0,Y 580.412,Z 923.055,A -85,B 0,C 180,E1 27419.341,E2 27419.341} C_VEL
LIN {X 0,Y 582.952,Z 903.733,A -85,B 0,C 180,E1 27417.704,E2 27417.704} C_VEL
LIN {X 0,Y 585.365,Z 885.323,A -85,B 0,C 180,E1 27416.338,E2 27416.338} C_VEL
LIN {X 0,Y 588.092,Z 863.106,A -85,B 0,C 180,E1 27414.923,E2 27414.923} C_VEL
LIN {X 0,Y 590.248,Z 843.978,A -85,B 0,C 180,E1 27413.877,E2 27413.877} C_VEL
LIN {X 0,Y 592.648,Z 820.801,A -85,B 0,C 180,E1 27412.806,E2 27412.806} C_VEL
LIN {X 0,Y 594.487,Z 799.765,A -85,B 0,C 180,E1 27412.005,E2 27412.005} C_VEL
LIN {X 0,Y 596.337,Z 775.952,A -85,B 0,C 180,E1 27411.271,E2 27411.271} C_VEL
LIN {X 0,Y 597.667,Z 752.906,A -85,B 0,C 180,E1 27410.742,E2 27410.742} C_VEL
LIN {X 0,Y 598.602,Z 729.735,A -85,B 0,C 180,E1 27410.351,E2 27410.351} C_VEL
LIN {X 0,Y 604.506,Z 476.957,A -85,B 0,C 180,E1 27406.951,E2 27406.951} C_VEL
LIN {X 0,Y 606.086,Z 407.629,A -85,B 0,C 180,E1 27405.996,E2 27405.996} C_VEL
LIN {X 0,Y 594.518,Z 388.483,A -85,B 0,C 180,E1 27404.636,E2 27404.636} C_VEL
LIN {X 0,Y 581.143,Z 368.229,A -85,B 0,C 180,E1 27402.983,E2 27402.983} C_VEL
LIN {X 0,Y 571.846,Z 355.177,A -85,B 0,C 180,E1 27401.774,E2 27401.774} C_VEL
LIN {X 0,Y 569.806,Z 352.204,A -85,B 0,C 180,E1 27401.498,E2 27401.498} C_VEL
LIN {X 0,Y 569.318,Z 350.274,A -85,B 0,C 180,E1 27401.194,E2 27401.194} C_VEL
LIN {X 0,Y 569.353,Z 350.309,A -85,B 0,C 180,E1 27397.928,E2 27397.928} C_VEL
LIN {X 0,Y 569.337,Z 350.272,A -85,B 0,C 180,E1 27394.805,E2 27394.805} C_VEL
LIN {X 0,Y 569.33,Z 350.299,A -85,B 0,C 180,E1 27391.558,E2 27391.558} C_VEL
LIN {X 0,Y 569.355,Z 350.299,A -85,B 0,C 180,E1 27388.534,E2 27388.534} C_VEL
LIN {X 0,Y 569.32,Z 350.299,A -85,B 0,C 180,E1 27385.246,E2 27385.246} C_VEL
LIN {X 0,Y 569.39,Z 350.293,A -85,B 0,C 180,E1 27382.074,E2 27382.074} C_VEL
LIN {X 0,Y 569.322,Z 350.31,A -85,B 0,C 180,E1 27378.854,E2 27378.854} C_VEL
LIN {X 0,Y 569.353,Z 350.307,A -85,B 0,C 180,E1 27375.587,E2 27375.587} C_VEL
LIN {X 0,Y 569.328,Z 350.307,A -85,B 0,C 180,E1 27372.579,E2 27372.579} C_VEL
LIN {X 0,Y 569.329,Z 350.303,A -85,B 0,C 180,E1 27369.196,E2 27369.196} C_VEL
LIN {X 0,Y 569.354,Z 350.297,A -85,B 0,C 180,E1 27366.15,E2 27366.15} C_VEL
LIN {X 0,Y 569.32,Z 350.309,A -85,B 0,C 180,E1 27362.919,E2 27362.919} C_VEL
LIN {X 0,Y 569.39,Z 350.306,A -85,B 0,C 180,E1 27359.698,E2 27359.698} C_VEL
LIN {X 0,Y 569.318,Z 350.298,A -85,B 0,C 180,E1 27356.476,E2 27356.476} C_VEL
LIN {X 0,Y 569.354,Z 350.291,A -85,B 0,C 180,E1 27353.243,E2 27353.243} C_VEL
LIN {X 0,Y 569.33,Z 350.313,A -85,B 0,C 180,E1 27350.15,E2 27350.15} C_VEL
LIN {X 0,Y 569.327,Z 350.309,A -85,B 0,C 180,E1 27346.802,E2 27346.802} C_VEL
LIN {X 0,Y 569.35,Z 350.295,A -85,B 0,C 180,E1 27343.785,E2 27343.785} C_VEL
LIN {X 0,Y 569.316,Z 350.293,A -85,B 0,C 180,E1 27340.507,E2 27340.507} C_VEL
LIN {X 0,Y 569.39,Z 350.292,A -85,B 0,C 180,E1 27337.382,E2 27337.382} C_VEL
LIN {X 0,Y 569.318,Z 350.312,A -85,B 0,C 180,E1 27334.179,E2 27334.179} C_VEL
LIN {X 0,Y 569.361,Z 350.307,A -85,B 0,C 180,E1 27330.892,E2 27330.892} C_VEL
LIN {X 0,Y 569.326,Z 350.313,A -85,B 0,C 180,E1 27327.835,E2 27327.835} C_VEL
LIN {X 0,Y 569.326,Z 350.314,A -85,B 0,C 180,E1 27324.405,E2 27324.405} C_VEL
LIN {X 0,Y 569.372,Z 350.309,A -85,B 0,C 180,E1 27321.235,E2 27321.235} C_VEL
LIN {X 0,Y 569.391,Z 350.343,A -85,B 0,C 180,E1 27318.946,E2 27318.946} C_VEL
LIN {X 0,Y 570.724,Z 353.923,A -85,B 0,C 180,E1 27318.394,E2 27318.394} C_VEL
LIN {X 0,Y 576.48,Z 367.303,A -85,B 0,C 180,E1 27316.326,E2 27316.326} C_VEL
LIN {X 0,Y 579.172,Z 373.346,A -85,B 0,C 180,E1 27315.464,E2 27315.464} C_VEL
LIN {X 0,Y 591.403,Z 392.552,A -85,B 0,C 180,E1 27313.925,E2 27313.925} C_VEL
LIN {X 0,Y 603.345,Z 412.578,A -85,B 0,C 180,E1 27312.501,E2 27312.501} C_VEL
LIN {X 0,Y 605.431,Z 416.842,A -85,B 0,C 180,E1 27312.249,E2 27312.249} C_VEL
LIN {X 0,Y 606.136,Z 421.288,A -85,B 0,C 180,E1 27312.117,E2 27312.117} C_VEL
LIN {X 0,Y 599.948,Z 683.573,A -85,B 0,C 180,E1 27308.578,E2 27308.578} C_VEL
LIN {X 0,Y 597.954,Z 766.151,A -85,B 0,C 180,E1 27307.454,E2 27307.454} C_VEL
LIN {X 0,Y 596.563,Z 791.68,A -85,B 0,C 180,E1 27306.948,E2 27306.948} C_VEL
LIN {X 0,Y 595.033,Z 813.35,A -85,B 0,C 180,E1 27306.368,E2 27306.368} C_VEL
LIN {X 0,Y 592.944,Z 838.191,A -85,B 0,C 180,E1 27305.516,E2 27305.516} C_VEL
LIN {X 0,Y 591.005,Z 857.874,A -85,B 0,C 180,E1 27304.69,E2 27304.69} C_VEL
LIN {X 0,Y 588.696,Z 879.583,A -85,B 0,C 180,E1 27303.622,E2 27303.622} C_VEL
LIN {X 0,Y 586.075,Z 901.435,A -85,B 0,C 180,E1 27302.334,E2 27302.334} C_VEL
LIN {X 0,Y 583.562,Z 922.052,A -85,B 0,C 180,E1 27300.932,E2 27300.932} C_VEL
LIN {X 0,Y 581.016,Z 941.713,A -85,B 0,C 180,E1 27299.371,E2 27299.371} C_VEL
LIN {X 0,Y 578.769,Z 959.142,A -85,B 0,C 180,E1 27297.805,E2 27297.805} C_VEL
LIN {X 0,Y 576.447,Z 977.418,A -85,B 0,C 180,E1 27295.92,E2 27295.92} C_VEL
LIN {X 0,Y 574.577,Z 992.602,A -85,B 0,C 180,E1 27294.139,E2 27294.139} C_VEL
LIN {X 0,Y 572.69,Z 1008.981,A -85,B 0,C 180,E1 27291.94,E2 27291.94} C_VEL
LIN {X 0,Y 571.321,Z 1021.701,A -85,B 0,C 180,E1 27289.977,E2 27289.977} C_VEL
LIN {X 0,Y 570.111,Z 1034.747,A -85,B 0,C 180,E1 27287.663,E2 27287.663} C_VEL
LIN {X 0,Y 569.304,Z 1044.734,A -85,B 0,C 180,E1 27285.588,E2 27285.588} C_VEL
LIN {X 0,Y 568.673,Z 1054.558,A -85,B 0,C 180,E1 27283.213,E2 27283.213} C_VEL
LIN {X 0,Y 568.282,Z 1062.131,A -85,B 0,C 180,E1 27280.947,E2 27280.947} C_VEL
LIN {X 0,Y 568.057,Z 1067.991,A -85,B 0,C 180,E1 27278.809,E2 27278.809} C_VEL
LIN {X 0,Y 567.95,Z 1073.173,A -85,B 0,C 180,E1 27276.266,E2 27276.266} C_VEL
LIN {X 0,Y 567.913,Z 1076.121,A -85,B 0,C 180,E1 27274.14,E2 27274.14} C_VEL
LIN {X 0,Y 567.903,Z 1077.97,A -85,B 0,C 180,E1 27271.917,E2 27271.917} C_VEL
LIN {X 0,Y 567.895,Z 1078.393,A -85,B 0,C 180,E1 27269.496,E2 27269.496} C_VEL
LIN {X 0,Y 567.907,Z 1077.493,A -85,B 0,C 180,E1 27267.376,E2 27267.376} C_VEL
LIN {X 0,Y 567.93,Z 1075.21,A -85,B 0,C 180,E1 27265.051,E2 27265.051} C_VEL
LIN {X 0,Y 567.987,Z 1071.101,A -85,B 0,C 180,E1 27262.617,E2 27262.617} C_VEL
LIN {X 0,Y 568.109,Z 1066.7,A -85,B 0,C 180,E1 27260.681,E2 27260.681} C_VEL
LIN {X 0,Y 568.39,Z 1059.935,A -85,B 0,C 180,E1 27258.328,E2 27258.328} C_VEL
LIN {X 0,Y 568.853,Z 1051.423,A -85,B 0,C 180,E1 27255.994,E2 27255.994} C_VEL
LIN {X 0,Y 569.527,Z 1041.953,A -85,B 0,C 180,E1 27253.791,E2 27253.791} C_VEL
LIN {X 0,Y 570.518,Z 1030.094,A -85,B 0,C 180,E1 27251.471,E2 27251.471} C_VEL
LIN {X 0,Y 571.654,Z 1018.64,A -85,B 0,C 180,E1 27249.523,E2 27249.523} C_VEL
LIN {X 0,Y 573.357,Z 1003.045,A -85,B 0,C 180,E1 27247.223,E2 27247.223} C_VEL
LIN {X 0,Y 575.004,Z 989.123,A -85,B 0,C 180,E1 27245.431,E2 27245.431} C_VEL
LIN {X 0,Y 577.244,Z 971.16,A -85,B 0,C 180,E1 27243.399,E2 27243.399} C_VEL
LIN {X 0,Y 579.352,Z 954.7,A -85,B 0,C 180,E1 27241.778,E2 27241.778} C_VEL
LIN {X 0,Y 581.832,Z 935.519,A -85,B 0,C 180,E1 27240.108,E2 27240.108} C_VEL
LIN {X 0,Y 584.245,Z 916.026,A -85,B 0,C 180,E1 27238.65,E2 27238.65} C_VEL
LIN {X 0,Y 586.781,Z 895.477,A -85,B 0,C 180,E1 27237.304,E2 27237.304} C_VEL
LIN {X 0,Y 589.214,Z 873.399,A -85,B 0,C 180,E1 27236.081,E2 27236.081} C_VEL
LIN {X 0,Y 591.294,Z 853.527,A -85,B 0,C 180,E1 27235.141,E2 27235.141} C_VEL
LIN {X 0,Y 593.524,Z 828.734,A -85,B 0,C 180,E1 27234.167,E2 27234.167} C_VEL
LIN {X 0,Y 595.213,Z 807.274,A -85,B 0,C 180,E1 27233.492,E2 27233.492} C_VEL
LIN {X 0,Y 596.905,Z 781.183,A -85,B 0,C 180,E1 27232.865,E2 27232.865} C_VEL
LIN {X 0,Y 597.85,Z 759.335,A -85,B 0,C 180,E1 27232.487,E2 27232.487} C_VEL
LIN {X 0,Y 603.083,Z 519.98,A -85,B 0,C 180,E1 27229.292,E2 27229.292} C_VEL
LIN {X 0,Y 605.254,Z 419.539,A -85,B 0,C 180,E1 27227.93,E2 27227.93} C_VEL
LIN {X 0,Y 604.046,Z 415.086,A -85,B 0,C 180,E1 27227.761,E2 27227.761} C_VEL
LIN {X 0,Y 589.277,Z 390.002,A -85,B 0,C 180,E1 27226.079,E2 27226.079} C_VEL
LIN {X 0,Y 578.551,Z 372.701,A -85,B 0,C 180,E1 27224.764,E2 27224.764} C_VEL
LIN {X 0,Y 572.143,Z 357.34,A -85,B 0,C 180,E1 27222.558,E2 27222.558} C_VEL
LIN {X 0,Y 569.373,Z 350.571,A -85,B 0,C 180,E1 27221.547,E2 27221.547} C_VEL
LIN {X 0,Y 569.371,Z 350.305,A -85,B 0,C 180,E1 27220.79,E2 27220.79} C_VEL
LIN {X 0,Y 569.319,Z 350.305,A -85,B 0,C 180,E1 27217.784,E2 27217.784} C_VEL
LIN {X 0,Y 569.353,Z 350.297,A -85,B 0,C 180,E1 27214.548,E2 27214.548} C_VEL
LIN {X 0,Y 569.322,Z 350.302,A -85,B 0,C 180,E1 27211.559,E2 27211.559} C_VEL
LIN {X 0,Y 569.331,Z 350.299,A -85,B 0,C 180,E1 27208.159,E2 27208.159} C_VEL
LIN {X 0,Y 569.361,Z 350.307,A -85,B 0,C 180,E1 27205.018,E2 27205.018} C_VEL
LIN {X 0,Y 569.319,Z 350.312,A -85,B 0,C 180,E1 27201.86,E2 27201.86} C_VEL
LIN {X 0,Y 569.373,Z 350.288,A -85,B 0,C 180,E1 27198.746,E2 27198.746} C_VEL
LIN {X 0,Y 569.317,Z 350.305,A -85,B 0,C 180,E1 27195.588,E2 27195.588} C_VEL
LIN {X 0,Y 569.381,Z 350.303,A -85,B 0,C 180,E1 27192.474,E2 27192.474} C_VEL
LIN {X 0,Y 569.318,Z 350.289,A -85,B 0,C 180,E1 27189.299,E2 27189.299} C_VEL
LIN {X 0,Y 569.354,Z 350.303,A -85,B 0,C 180,E1 27186.049,E2 27186.049} C_VEL
LIN {X 0,Y 569.335,Z 350.302,A -85,B 0,C 180,E1 27182.919,E2 27182.919} C_VEL
LIN {X 0,Y 569.324,Z 350.288,A -85,B 0,C 180,E1 27179.597,E2 27179.597} C_VEL
LIN {X 0,Y 569.366,Z 350.307,A -85,B 0,C 180,E1 27176.476,E2 27176.476} C_VEL
LIN {X 0,Y 569.317,Z 350.298,A -85,B 0,C 180,E1 27173.242,E2 27173.242} C_VEL
LIN {X 0,Y 569.378,Z 350.295,A -85,B 0,C 180,E1 27170.09,E2 27170.09} C_VEL
LIN {X 0,Y 569.323,Z 350.309,A -85,B 0,C 180,E1 27166.905,E2 27166.905} C_VEL
LIN {X 0,Y 569.355,Z 350.29,A -85,B 0,C 180,E1 27163.681,E2 27163.681} C_VEL
LIN {X 0,Y 569.335,Z 350.308,A -85,B 0,C 180,E1 27160.579,E2 27160.579} C_VEL
LIN {X 0,Y 569.33,Z 350.313,A -85,B 0,C 180,E1 27157.225,E2 27157.225} C_VEL
LIN {X 0,Y 569.372,Z 350.288,A -85,B 0,C 180,E1 27154.045,E2 27154.045} C_VEL
LIN {X 0,Y 569.321,Z 350.295,A -85,B 0,C 180,E1 27150.89,E2 27150.89} C_VEL
LIN {X 0,Y 569.385,Z 350.3,A -85,B 0,C 180,E1 27147.734,E2 27147.734} C_VEL
LIN {X 0,Y 569.325,Z 350.311,A -85,B 0,C 180,E1 27144.578,E2 27144.578} C_VEL
LIN {X 0,Y 569.36,Z 350.309,A -85,B 0,C 180,E1 27141.303,E2 27141.303} C_VEL
LIN {X 0,Y 569.333,Z 350.316,A -85,B 0,C 180,E1 27138.27,E2 27138.27} C_VEL
LIN {X 0,Y 569.331,Z 350.266,A -85,B 0,C 180,E1 27134.911,E2 27134.911} C_VEL
LIN {X 0,Y 569.339,Z 350.369,A -85,B 0,C 180,E1 27134.23,E2 27134.23} C_VEL
